//Error FB instances
EL5021_Error(
    En                  := TRUE,
    iTerminal_ID        := iTerminal_ID,
    bWcState            := WcState_WcState,
    uiInfoData_State    := InfoData_State,
    pErrorSystem        := ErrorSystem,
    bError => bError,
);

IF bError THEN
    sErrorMessage:=EL5021_Error.ErrorData.sErrorMessage;
ELSE
	sErrorMessage:='';
END_IF

END_FUNCTION_BLOCK

// ---- POUs/Common/Hardware/EtherCAT_Terminals/Communication/EL6695.TcPOU
//EL6695 | EtherCAT bridge termina
FUNCTION_BLOCK EL6695

VAR_INPUT
    En: BOOL;
    iTerminal_ID : INT;
    ErrorSystem : POINTER TO ST_ErrorSystem;
END_VAR

VAR_OUTPUT
    EnO: BOOL;
    bError: BOOL;
	sErrorMessage       : STRING;
END_VAR

VAR
    WcState_WcState AT %I* : BOOL := FALSE;
    InfoData_State  AT %I* : UINT := 0;

    //FB-s
    EL6695_Error    : FB_TerminalError;
END_VAR

(*
* TODO: Test on hardware
*)

EnO:=En;

EL6695_Error(
    En := TRUE,
    iTerminal_ID := iTerminal_ID,
    bWcState := FALSE,
    uiInfoData_State := InfoData_State,
    pErrorSystem := ErrorSystem,
    bError => bError,
);

IF bError THEN
	sErrorMessage:=EL6695_Error.ErrorData.sErrorMessage;
ELSE
	sErrorMessage:='';
END_IF

END_FUNCTION_BLOCK

// ---- POUs/Common/Hardware/EtherCAT_Terminals/Digital_Outputs/EL2032.TcPOU
// EL2032 | 2-channel digital output terminal 24 V DC, 2 A
FUNCTION_BLOCK EL2032

VAR_INPUT
    En: BOOL;
    iTerminal_ID : INT;
    ErrorSystem : POINTER TO ST_ErrorSystem;
END_VAR

VAR_OUTPUT
    EnO: BOOL;
    bError: BOOL;
	sErrorMessage       : STRING;
END_VAR

VAR
    WcState_WcState AT %I* : BOOL := FALSE;
    InfoData_State  AT %I* : UINT := 0;

    //FB-s
    EL2032_Error    : FB_TerminalError;
END_VAR

(*
* TODO: Test on hardware
*)

EnO:=En;

EL2032_Error(
    En := TRUE,
    iTerminal_ID := iTerminal_ID,
    bWcState := FALSE,
    uiInfoData_State := InfoData_State,
    pErrorSystem := ErrorSystem,
    bError => bError,
);

IF bError THEN
	sErrorMessage:=EL2032_Error.ErrorData.sErrorMessage;
ELSE
	sErrorMessage:='';
END_IF

END_FUNCTION_BLOCK

// ---- POUs/Common/Hardware/EtherCAT_Terminals/System/EK1110.TcPOU
FUNCTION_BLOCK EK1110

VAR_INPUT
    En              : BOOL;
    iTerminal_ID    : INT;
    ErrorSystem     : POINTER TO ST_ErrorSystem;
END_VAR

VAR_OUTPUT
    EnO     : BOOL;
    bError  : BOOL;
	sErrorMessage       : STRING;
END_VAR

VAR
    InfoData_State  AT %I*  : UINT;
    
    //FB-s
    EK1110_Error    : FB_TerminalError;
END_VAR

(*
* TODO: DONE!
*)
EnO:=En;

//Error FB instance
EK1110_Error(
    En                  := TRUE,
    iTerminal_ID        := iTerminal_ID,
    bWcState            := FALSE,
    uiInfoData_State    := InfoData_State,
    pErrorSystem        := ErrorSystem,
    bError              => bError,
);

IF bError THEN
	sErrorMessage:=EK1110_Error.ErrorData.sErrorMessage;
ELSE
	sErrorMessage:='';
END_IF

END_FUNCTION_BLOCK

// ---- POUs/Common/Hardware/EtherCAT_Terminals/Drives/indraDrive.TcPOU
//Rexroth indradrive
FUNCTION_BLOCK indraDrive

VAR_INPUT
    En: BOOL;
    iTerminal_ID : INT;
    ErrorSystem : POINTER TO ST_ErrorSystem;
END_VAR

VAR_OUTPUT
    EnO: BOOL;
    bError: BOOL;
	sErrorMessage       : STRING;
END_VAR

VAR
    WcState_WcState AT %I* : BOOL := FALSE;
    InfoData_State  AT %I* : UINT := 0;

    //FB-s
    indraDrive_Error    : FB_TerminalError;
END_VAR

(*
* TODO: Test on hardware
*)

EnO:=En;

indraDrive_Error(
    En := TRUE,
    iTerminal_ID := iTerminal_ID,
    bWcState := FALSE,
    uiInfoData_State := InfoData_State,
    pErrorSystem := ErrorSystem,
    bError => bError,
);

IF bError THEN
	sErrorMessage:=indraDrive_Error.ErrorData.sErrorMessage;
ELSE
	sErrorMessage:='';
END_IF

END_FUNCTION_BLOCK

// ---- POUs/Common/Hardware/EtherCAT_Terminals/Drives/iPOS8020.TcPOU
//Technosoft iPOS8020
FUNCTION_BLOCK iPOS8020

VAR_INPUT
    En: BOOL;
    iTerminal_ID : INT;
    ErrorSystem : POINTER TO ST_ErrorSystem;
END_VAR

VAR_OUTPUT
    EnO: BOOL;
    bError: BOOL;
	sErrorMessage       : STRING;
END_VAR

VAR
    WcState_WcState AT %I* : BOOL := FALSE;
    InfoData_State  AT %I* : UINT := 0;

    //FB-s
    iPOS8020_Error    : FB_TerminalError;
END_VAR

(*
* TODO: Test on hardware
*)

EnO:=En;

iPOS8020_Error(
    En := TRUE,
    iTerminal_ID := iTerminal_ID,
    bWcState := FALSE,
    uiInfoData_State := InfoData_State,
    pErrorSystem := ErrorSystem,
    bError => bError,
);

IF bError THEN
	sErrorMessage:=iPOS8020_Error.ErrorData.sErrorMessage;
ELSE
	sErrorMessage:='';
END_IF

END_FUNCTION_BLOCK

// ---- POUs/Bridge Terminal/TSCS_Bridge_Inputs.TcPOU
PROGRAM TSCS_Bridge_Inputs	
(* Inputs from TSCS PLC to TDU PLC*)
VAR
	// Function Blocks
	BYTE_TO_BITS_10: OSCAT_BYTE_TO_BITS; // Interface for TSCS Byte 0 - Boolean inputs
	BYTE_TO_BITS_11: OSCAT_BYTE_TO_BITS; // Interface for TSCS Byte 1 - Boolean inputs
	BYTE_TO_BITS_12: OSCAT_BYTE_TO_BITS; // Interface for TSCS Byte 2 - Boolean inputs
	BYTE_TO_BITS_13: OSCAT_BYTE_TO_BITS; // Interface for TSCS Byte 3 - Boolean inputs
	fb_Bridge_Real_Inputs_0 : FB_Bridge_Inputs_Real; // Interface for TSCS real signals
	fb_Bridge_Real_Inputs_1 : FB_Bridge_Inputs_Real; // Interface for TMS real signals
	
	// Test Signal
	TDU_TestSignal_RB : REAL;	// Diagnostic signal readback (TDU -> TSCS ->TDU)
		
	// TSCS signals (as example)
	Lube_MainBearing_Act : BOOL; 		// Main bearing lubrication active
	TSCS_State : INT; 					// Target System Operation Mode [0=Off, 1=Normal Operation, 2=Maintenance]
	Lube_MainBearing_FlowRate : REAL; 	// Main bearing lubrication flow rate [mL/min]
END_VAR

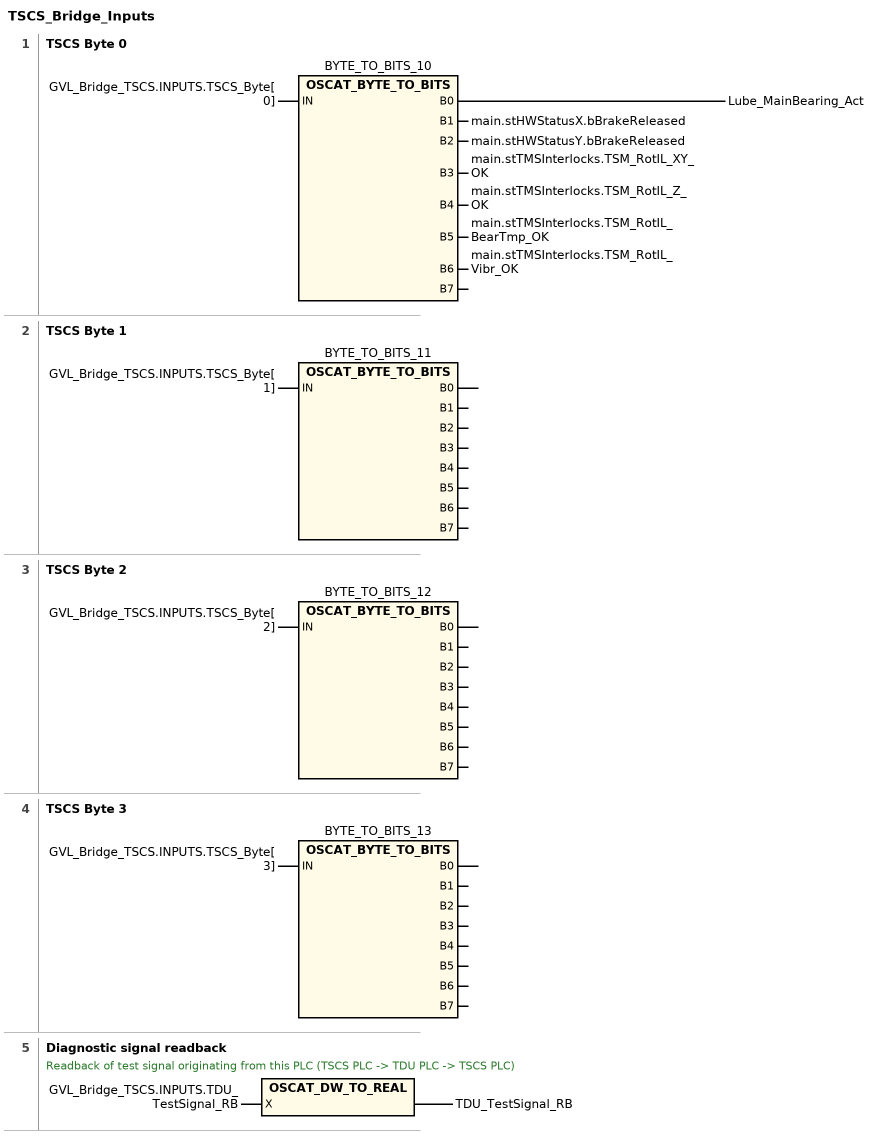
// NETWORK 1: TSCS Byte 0
BYTE_TO_BITS_10(
    IN := GVL_Bridge_TSCS.INPUTS.TSCS_Byte[0],
    B1 => main.stHWStatusX.bBrakeReleased,
    B2 => main.stHWStatusY.bBrakeReleased,
    B3 => main.stTMSInterlocks.TSM_RotIL_XY_OK,
    B4 => main.stTMSInterlocks.TSM_RotIL_Z_OK,
    B5 => main.stTMSInterlocks.TSM_RotIL_BearTmp_OK,
    B6 => main.stTMSInterlocks.TSM_RotIL_Vibr_OK); // OSCAT_BYTE_TO_BITS
Lube_MainBearing_Act := BYTE_TO_BITS_10.B0;

// NETWORK 2: TSCS Byte 1
BYTE_TO_BITS_11(IN := GVL_Bridge_TSCS.INPUTS.TSCS_Byte[1]); // OSCAT_BYTE_TO_BITS

// NETWORK 3: TSCS Byte 2
BYTE_TO_BITS_12(IN := GVL_Bridge_TSCS.INPUTS.TSCS_Byte[2]); // OSCAT_BYTE_TO_BITS

// NETWORK 4: TSCS Byte 3
BYTE_TO_BITS_13(IN := GVL_Bridge_TSCS.INPUTS.TSCS_Byte[3]); // OSCAT_BYTE_TO_BITS

// NETWORK 5: Diagnostic signal readback
// Readback of test signal originating from this PLC (TSCS PLC -> TDU PLC -> TSCS PLC)
TDU_TestSignal_RB := OSCAT_DW_TO_REAL(X := GVL_Bridge_TSCS.INPUTS.TDU_TestSignal_RB);

END_PROGRAM

// ---- POUs/Bridge Terminal/FBs/OSCAT_BYTE_TO_BITS.TcPOU
FUNCTION_BLOCK OSCAT_BYTE_TO_BITS
// E. Foy (2021-08-30): Copied from OSCAT library.
VAR_INPUT
	IN: BYTE;
END_VAR
VAR_OUTPUT
	B0: BOOL;
	B1: BOOL;
	B2: BOOL;
	B3: BOOL;
	B4: BOOL;
	B5: BOOL;
	B6: BOOL;
	B7: BOOL;
END_VAR


(*
version 1.1	16. mar. 2008
programmer 	hugo
tested by		tobias

this Function Block extracts the 8 Bits from a byte


*)

B0 := IN.0;
B1 := IN.1;
B2 := IN.2;
B3 := IN.3;
B4 := IN.4;
B5 := IN.5;
B6 := IN.6;
B7 := IN.7;

(* revision history
hm		4. aug 2006	rev 1.0
	original version

hm		16. mar 2008	rev 1.1
	renamed from byte_to_bit to byte_to_bits for compatibility reasons

*)

END_FUNCTION_BLOCK

// ---- POUs/Bridge Terminal/FBs/FB_Bridge_Inputs_Real.TcPOU
FUNCTION_BLOCK FB_Bridge_Inputs_Real
// Interface with 20 ports. Converts UDINT to REAL (32 bits)
VAR_INPUT
	I00 : UDINT := 0;	// Input real 00
	I01 : UDINT := 0;	// Input real 01
	I02 : UDINT := 0;	// Input real 02
	I03 : UDINT := 0;	// Input real 03
	I04 : UDINT := 0;	// Input real 04
	I05 : UDINT := 0;	// Input real 05
	I06 : UDINT := 0;	// Input real 06
	I07 : UDINT := 0;	// Input real 07
END_VAR
VAR_OUTPUT
	Q00 : REAL;
	Q01 : REAL;
	Q02 : REAL;
	Q03 : REAL;
	Q04 : REAL;
	Q05 : REAL;
	Q06 : REAL;
	Q07 : REAL;
END_VAR
VAR
END_VAR

Q00 := OSCAT_DW_TO_REAL(I00);
Q01 := OSCAT_DW_TO_REAL(I01);
Q02 := OSCAT_DW_TO_REAL(I02);
Q03 := OSCAT_DW_TO_REAL(I03);
Q04 := OSCAT_DW_TO_REAL(I04);
Q05 := OSCAT_DW_TO_REAL(I05);
Q06 := OSCAT_DW_TO_REAL(I06);
Q07 := OSCAT_DW_TO_REAL(I07);

END_FUNCTION_BLOCK

// ---- POUs/Bridge Terminal/FBs/OSCAT_DW_TO_REAL.TcPOU
FUNCTION OSCAT_DW_TO_REAL : REAL
// E. Foy (2021-08-30): Copied from OSCAT library.
VAR_INPUT
	X : DWORD;
END_VAR
VAR
	pt : POINTER TO REAL;
END_VAR

(*
version 1.0	18. apr. 2008
programmer 	hugo
tested by		tobias

this function converts a DWORD to REAL in a bitwise manner.
*)

pt := ADR(X);
OSCAT_DW_TO_REAL := pt^;

(* revision history
hm	18. apr. 2008
	original version

*)

END_FUNCTION

// ---- POUs/Bridge Terminal/TSCS_Bridge_Diagnostic.TcPOU
PROGRAM TSCS_Bridge_Diagnostic
(*Generates a test signal for the bridge terminal then compares it against a readback signal*)
VAR
	TestSignal : REAL;
	
	TDU_TestSignal_Delay :REAL := 0; // Number of counts behind the TDU TestSignal
	TMS_TestSignal_Delay :REAL := 0; // Number of counts behind the TMS TestSignal 
	
	// Parameters
	CountRate : REAL := 1.0; // ms per cycle (e.g. 1.0 for a 1ms excution rate)
	Signal_HL : REAL := 1000; // Signal High Limit
	Signal_LL : REAL := -1000; // Signal Low Limit
 
	RS_0: RS;	// Counter state (Set = Count-DOWN active)
END_VAR
VAR // added by the converter: edge detectors and wires of the graphical bodies
    _rt1, _rt2 : R_TRIG;
END_VAR

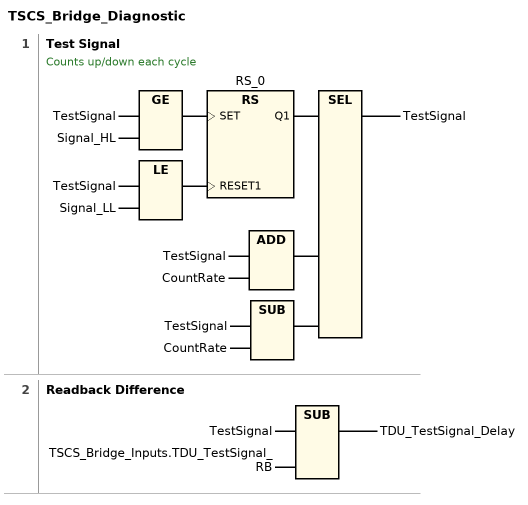
// NETWORK 1: Test Signal
// Counts up/down each cycle
_rt1(CLK := TestSignal >= Signal_HL);
_rt2(CLK := TestSignal <= Signal_LL);
RS_0(SET := _rt1.Q, RESET1 := _rt2.Q); // RS
TestSignal := SEL(RS_0.Q1, TestSignal + CountRate, TestSignal - CountRate);

// NETWORK 2: Readback Difference
TDU_TestSignal_Delay := TestSignal - TSCS_Bridge_Inputs.TDU_TestSignal_RB;

END_PROGRAM

// ---- POUs/Bridge Terminal/TSCS_Bridge_Outputs.TcPOU
PROGRAM TSCS_Bridge_Outputs
(*Outputs from TDU PLC to TSCS PLC*)
VAR
	// Function Blocks
	fb_Bridge_Outputs_Real_0 : FB_Bridge_Outputs_Real; // Interface for TDU real outputs
	
	// Signal Conversions
	rActPos : REAL; // Rotation system - Actual Position [deg]
	rActVel : REAL; // Rotation system - Actual Velocity [rpm]
	rSetVelRaw : REAL; //Rotation system - Velocity setpoint raw [rpm] 
	
END_VAR

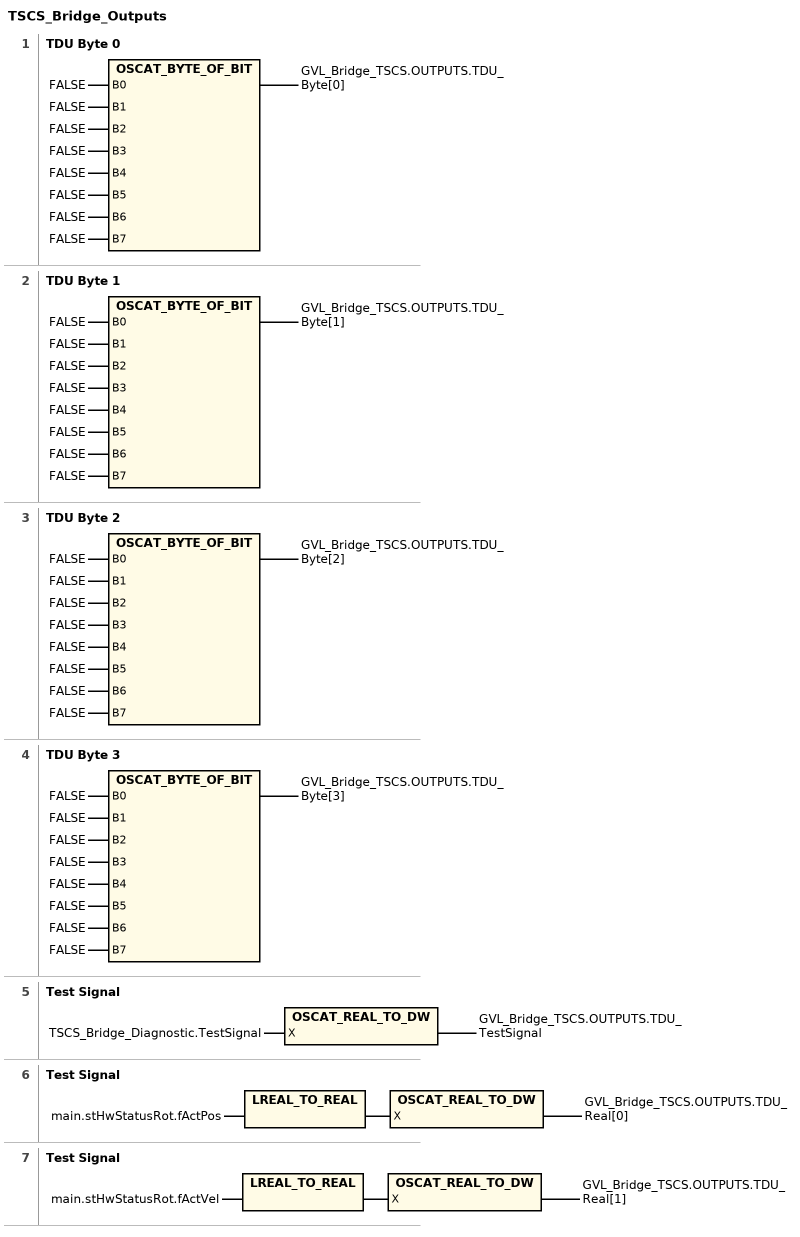
// NETWORK 1: TDU Byte 0
GVL_Bridge_TSCS.OUTPUTS.TDU_Byte[0] := OSCAT_BYTE_OF_BIT(B0 := FALSE, B1 := FALSE, B2 := FALSE, B3 := FALSE, B4 := FALSE, B5 := FALSE, B6 := FALSE, B7 := FALSE);

// NETWORK 2: TDU Byte 1
GVL_Bridge_TSCS.OUTPUTS.TDU_Byte[1] := OSCAT_BYTE_OF_BIT(B0 := FALSE, B1 := FALSE, B2 := FALSE, B3 := FALSE, B4 := FALSE, B5 := FALSE, B6 := FALSE, B7 := FALSE);

// NETWORK 3: TDU Byte 2
GVL_Bridge_TSCS.OUTPUTS.TDU_Byte[2] := OSCAT_BYTE_OF_BIT(B0 := FALSE, B1 := FALSE, B2 := FALSE, B3 := FALSE, B4 := FALSE, B5 := FALSE, B6 := FALSE, B7 := FALSE);

// NETWORK 4: TDU Byte 3
GVL_Bridge_TSCS.OUTPUTS.TDU_Byte[3] := OSCAT_BYTE_OF_BIT(B0 := FALSE, B1 := FALSE, B2 := FALSE, B3 := FALSE, B4 := FALSE, B5 := FALSE, B6 := FALSE, B7 := FALSE);

// NETWORK 5: Test Signal
GVL_Bridge_TSCS.OUTPUTS.TDU_TestSignal := OSCAT_REAL_TO_DW(X := TSCS_Bridge_Diagnostic.TestSignal);

// NETWORK 6: Test Signal
GVL_Bridge_TSCS.OUTPUTS.TDU_Real[0] := OSCAT_REAL_TO_DW(X := LREAL_TO_REAL(main.stHwStatusRot.fActPos));

// NETWORK 7: Test Signal
GVL_Bridge_TSCS.OUTPUTS.TDU_Real[1] := OSCAT_REAL_TO_DW(X := LREAL_TO_REAL(main.stHwStatusRot.fActVel));

END_PROGRAM

// ---- POUs/Bridge Terminal/FBs/FB_Bridge_Outputs_Real.TcPOU
FUNCTION_BLOCK FB_Bridge_Outputs_Real
// Interface with 20 ports. Converts REAL to UDINT (32 bits)
VAR_INPUT
	I00 : REAL := 0;
	I01 : REAL := 0;
	I02 : REAL := 0;
	I03 : REAL := 0;
	I04 : REAL := 0;
	I05 : REAL := 0;
	I06 : REAL := 0;
	I07 : REAL := 0;
END_VAR
VAR_OUTPUT
	Q00 : UDINT;
	Q01 : UDINT;
	Q02 : UDINT;
	Q03 : UDINT;
	Q04 : UDINT;
	Q05 : UDINT;
	Q06 : UDINT;
	Q07 : UDINT;
END_VAR
VAR
END_VAR

Q00 := OSCAT_REAL_TO_DW(I00);
Q01 := OSCAT_REAL_TO_DW(I01);
Q02 := OSCAT_REAL_TO_DW(I02);
Q03 := OSCAT_REAL_TO_DW(I03);
Q04 := OSCAT_REAL_TO_DW(I04);
Q05 := OSCAT_REAL_TO_DW(I05);
Q06 := OSCAT_REAL_TO_DW(I06);
Q07 := OSCAT_REAL_TO_DW(I07);

END_FUNCTION_BLOCK

// ---- POUs/Bridge Terminal/FBs/OSCAT_REAL_TO_DW.TcPOU
FUNCTION OSCAT_REAL_TO_DW : DWORD
// E. Foy (2021-08-30): Copied from OSCAT library.
VAR_INPUT
	X : REAL;
END_VAR
VAR
	pt : POINTER TO DWORD;
END_VAR

(*
version 1.0	18. apr. 2008
programmer 	hugo
tested by		tobias

this function converts a 32 Bit Real to a dword in a bitwise manner.
*)

pt := ADR(X);
OSCAT_REAL_TO_DW := pt^;

(* revision history
hm	18. apr. 2008
	original version

*)

END_FUNCTION

// ---- POUs/Bridge Terminal/FBs/OSCAT_BYTE_OF_BIT.TcPOU
FUNCTION OSCAT_BYTE_OF_BIT : BYTE
// E. Foy (2021-08-30): Copied from OSCAT library.
VAR_INPUT
	B0:BOOL;
	B1:BOOL;
	B2:BOOL;
	B3:BOOL;
	B4:BOOL;
	B5:BOOL;
	B6:BOOL;
	B7:BOOL;
END_VAR

(*
version 1.1	 18. feb 2006
programmer 	hugo
tested by		tobias

this function creates a byte from 8 individual bits

*)

OSCAT_BYTE_OF_BIT := SHL(SHL(SHL(SHL(SHL(SHL(SHL(BOOL_TO_BYTE(B7),1) OR BOOL_TO_BYTE(B6),1) OR BOOL_TO_BYTE(B5),1) OR BOOL_TO_BYTE(B4),1)
	OR BOOL_TO_BYTE(B3),1) OR BOOL_TO_BYTE(B2),1) OR BOOL_TO_BYTE(B1),1) OR BOOL_TO_BYTE(B0);


(* revision history

hm	4. aug 2006		rev 1.0
	original version

hm	18. feb. 2008	rev 1.1
	improved performance

*)

END_FUNCTION

// ---- POUs/MAIN_NORMAL_MOTION.TcPOU
PROGRAM MAIN_NORMAL_MOTION
VAR
    sVersion: STRING := '1.0.0';

    //hmiAxisSelection: INT := 1; //Not possible to use local hmi variables for array indexes

//Startup, Shutdown and UPS
    fbUPS: FB_S_UPS_CX51x0;
    eUpsMode: E_S_UPS_Mode := eSUPS_WrPersistData_Shutdown;
    eStartUp: (eColdStart, eReadAxisFeedbackType, eCheckReadDone, eExecuteRestore, eCheckRestore, eFinishRestore);
    bPositionRestoreDone: BOOL := FALSE;
    bRestoreExecute: BOOL := FALSE;
    bExecuteReadEncRefSys: BOOL := FALSE;
    nRetry: INT;
    iAxes : UINT; //index for for loops in Position recovery actions
    afbReadEncRefSys: ARRAY [1..GVL_APP.nAXIS_NUM] OF MC_ReadParameter;
    afbRestorePosition: ARRAY [1..GVL_APP.nAXIS_NUM] OF MC_SetPosition;
    fbGetDeviceIdentification: FB_GetDeviceIdentification;
END_VAR

VAR PERSISTENT
    bRestoreOnStartup: BOOL;
END_VAR

// Block PILS
GVL.bLocalMode:=TRUE;

POSITION_RECOVERY();
AXES();
PROG();

ACTION AXES:
//Get task index for Axes parameters initialization.
GVL.fbGetCurTaskIndex();

//Create an stAxisStruct for every axis in the project.
FOR GVL.iAxis := 1 TO GVL_APP.nAXIS_NUM DO
    Main.afbAxes[GVL.iAxis](stAxisStruct := GVL.astAxes[GVL.iAxis]);
END_FOR
END_ACTION

ACTION CHECK_UPS:
fbUPS(eUpsMode := eUpsMode);

IF eGlobalSUpsState = eSUPS_PowerFailure THEN
    //first cycle of powerfailure
    //execute code that should only be done once with each powerfailure, i.e. increase powerfailure counter
    bRestoreOnStartup := TRUE;
    STORE_PERSISTENT();
    RETURN;
ELSIF eGlobalSUpsState <> eSUPS_PowerOK THEN
    //next cycles of powerfailure
    //skip regular code execution for the remaining cycles of the powerfailure/writing of persistent data/quick shutdown...
    RETURN;
END_IF
END_ACTION

ACTION POSITION_RECOVERY:
fbGetDeviceIdentification(bExecute := TRUE);
IF (fbGetDeviceIdentification.stDevIdent.strHardwareSerialNo <> '0') THEN
    CHECK_UPS();
    RESTORE_POSITIONS();
END_IF
END_ACTION

ACTION PROG:
//Call the programs that are defined in the "Application Specific" folder.
//Create as many programs in that folder as axes and applications you have or need

//Axes initial parameters and program
//Axis_Template();
Axis_1();
Axis_2();
Axis_3();

//Application program calls
//Application_Template();
END_ACTION

ACTION RESTORE_POSITIONS:
//This ACT will restore the position of an incremental axis on startup with the act position it read before losing power.
//It checks the type of axis, 0=incremental, and that the axis was stationary at shut down.
//Because 0 equates to incremental we also need to check that the data is valid, otherwise by default it would restore all axes.
//By default an axis will not restore the position unless it is set to opt-in, i.e. GVL.aAxes[iAxes].stConfig.eRestorePosition is non-zero.
//This needs to be initialised somewhere in TwinCAT code otherwise it will not be available at start up.
//A restore will only be performed on a loss of power, this code shouldn't make any changes on a reset cold, a rest origin or a download.
//There is a enum to allow for different types of restore modes, currently only one is implemented.
//0 'DontRestore'
//1 'RestoreWithoutHome' -restores the position using a set position fb and does not set the home bit in the axis struct.
//Note from Beckhoff: "A maximum of 1 MB persistent data can be reliably saved over the entire service life."

IF bRestoreOnStartup AND eGlobalSUpsState = eSUPS_PowerOK THEN
    bRestoreOnStartup := FALSE;
    bRestoreExecute := TRUE;
END_IF

//Upon startup bPositionRestoreDone will be set to FALSE, after successfully completing the following code it will be set TRUE
//and should stay TRUE for the rest of the time the PLC is operational, thus this routine should only be completed once.
IF bRestoreExecute AND NOT bPositionRestoreDone THEN
    //Cycle through function blocks that read the encoder reference system i.e. whether axis is incremental or absolute
    //Result stored in Value, 0=Inc 1=Abs, execute set during the case statement
    FOR iAxes := 1 TO GVL_APP.nAXIS_NUM DO
        afbReadEncRefSys[iAxes](
          Axis := GVL.astAxes[iAxes].Axis,
          Enable := bExecuteReadEncRefSys,
          ParameterNumber := MC_AxisParameter.AxisEncoderReferenceSystem,
          ReadMode := E_READMODE.READMODE_ONCE);
    END_FOR

    //Cycle through set position function blocks for each axis
    FOR iAxes := 1 TO GVL_APP.nAXIS_NUM DO
        afbRestorePosition[iAxes](
         Axis := GVL.astAxes[iAxes].Axis,
         Position := astAxesPersistent[iAxes].fPositionAtShutdown);
    END_FOR

    CASE eStartUp OF
        eColdStart:
        //First cycle of the PLC, do nothing just give one cycle for variables to initialise
            IF NOT bPositionRestoreDone THEN
                eStartUp := eReadAxisFeedbackType;
                nRetry := 0;
            END_IF

        eReadAxisFeedbackType:
        //Exectute the function blocks to read the encoder reference system (0=inc OR 1=ABS)
            bExecuteReadEncRefSys := TRUE;
            eStartUp := eCheckReadDone;

        eCheckReadDone:
        //Check the encoder reference system has been read for all axis -> if busy then continue with PLC cycle and check again next time.
        //If afbReadEncRefSys not started then go back a step.
        //If any axes result in an error the code will get stuck here, this happens if GVL_APP.nAXIS_NUM is not set correctly
            FOR iAxes := 1 TO GVL_APP.nAXIS_NUM DO
                IF afbReadEncRefSys[iAxes].Valid = FALSE THEN
                    IF afbReadEncRefSys[iAxes].Busy = TRUE THEN
                        //Exit MAIN.STARTUP Action and wait till next cycle, needs to cycle through whole program in order for data to update
                        RETURN;
                    ELSE
                        //Sometimes the code gets here and the afbReadEncRefSys[iAxes] misses the rising edge. If  the code gets here it means
                        //valid=FALSE and .busy=FALSE which indicateds the FB probably hasn't started and thus needs to see a rising edge.
                        //Set execute to low, Exit MAIN.STARTUP and go back a step in the CASE statement.
                        bExecuteReadEncRefSys := FALSE;
                        eStartUp := eReadAxisFeedbackType;
                        nRetry := nRetry + 1; //counter used for troubleshooting to see how many cycles it takes before afbReadEncRefSys function blocks are read correctly
                        RETURN;
                    END_IF
                END_IF
            END_FOR
            //If the code gets here all axes either have .valid=TRUE for all axes
            eStartUp := eExecuteRestore;

        eExecuteRestore:
        //Execute position restore by setting afbRestorePosition.execute = TRUE
            FOR iAxes := 1 TO GVL_APP.nAXIS_NUM DO
                IF afbReadEncRefSys[iAxes].Valid = TRUE AND afbReadEncRefSys[iAxes].Value = 0 AND NOT(astAxesPersistent[iAxes].bMovingAtShutdown) THEN
                    IF GVL.astAxes[iAxes].stConfig.eRestorePosition = E_RestorePosition.eRestoreWithoutHome THEN
                        afbRestorePosition[iAxes].Execute := TRUE;
                    END_IF
                END_IF
            END_FOR
            eStartUp := eCheckRestore;

        eCheckRestore:
        //Check the set position fbs are finished
        //Nothing actually happens if the restore is not done, the code just returns from here each cycle and the
        //bPositionRestoreDone will never get set to TRUE and will take up cycle time
            FOR iAxes := 1 TO GVL_APP.nAXIS_NUM DO
                IF afbReadEncRefSys[iAxes].Valid = TRUE AND afbReadEncRefSys[iAxes].Value = 0 AND NOT(astAxesPersistent[iAxes].bMovingAtShutdown) THEN
                    IF GVL.astAxes[iAxes].stConfig.eRestorePosition = E_RestorePosition.eRestoreWithoutHome THEN
                        IF NOT afbRestorePosition[iAxes].Done THEN
                            RETURN;
                        END_IF
                    END_IF
                END_IF
            END_FOR
            eStartUp := eFinishRestore;

        eFinishRestore:
        //Remove execute = TRUE for afbRestorePosition
            FOR iAxes := 1 TO GVL_APP.nAXIS_NUM DO
                afbRestorePosition[iAxes].Execute := FALSE;
            END_FOR
            bPositionRestoreDone := TRUE;
            bRestoreExecute := FALSE;
    END_CASE
END_IF
END_ACTION

ACTION STORE_PERSISTENT:
FOR iAxes := 1 TO GVL_APP.nAXIS_NUM DO
    astAxesPersistent[iAxes].fPositionAtShutdown := GVL.astAxes[iAxes].Axis.NcToPlc.ActPos;
    IF GVL.astAxes[iAxes].Axis.NcToPlc.ActVelo <> 0 THEN
        astAxesPersistent[iAxes].bMovingAtShutdown := TRUE;
    ELSE
        astAxesPersistent[iAxes].bMovingAtShutdown := FALSE;
    END_IF
    astAxesPersistent[iAxes].bMovingAtShutdown := astAxesPersistent[iAxes].bMovingAtShutdown OR GVL.astAxes[iAxes].Axis.Status.Moving;
END_FOR
END_ACTION

END_PROGRAM

// ---- POUs/Application_Specific/Axes/Axis_1.TcPOU
PROGRAM Axis_1
VAR
    bLimitPowerAxis1 AT %Q*: BOOL := TRUE;
END_VAR
VAR // added by the converter: edge detectors and wires of the graphical bodies
    _w1, _w2 : BOOL;
END_VAR

//Initial parameters of an Axis
IF _TaskInfo[fbGetCurTaskIndex.index].FirstCycle THEN
    //Initial default values:
    GVL.astAxes[1].stConfig.eHomeSeq := 0;
    GVL.astAxes[1].stConfig.fHomePosition := 0.0;
    GVL.astAxes[1].stConfig.fHomeFinishDistance := 0.0;
END_IF

ACT_1_Interlock();

// Brake control from GUI
// main.stHWStatusX.bBrakeReleased:=main.stHWControlX.bBrakeReleaseCmd;

// Enable Cmd from GUI
GVL.astAxes[1].stControl.bEnable:=main.stHWControlX.bEnable;
main.stHWStatusX.bEnabled:=GVL.astAxes[1].stStatus.bEnabled;

// Trigger Abs movement from GUI
IF main.stHWControlX.bExecuteAbsPos  AND NOT GVL.astAxes[1].stStatus.bBusy THEN
  GVL.astAxes[1].stControl.eCommand:=E_MotionFunctions.eMoveAbsolute;
  GVL.astAxes[1].stControl.bExecute:=TRUE;
  main.stHWControlX.bExecuteAbsPos:=FALSE;
END_IF

// Trigger Const Velo movement from GUI
IF main.stHWControlX.bExecuteConstVelo AND NOT GVL.astAxes[1].stStatus.bBusy THEN
  GVL.astAxes[1].stControl.eCommand:=E_MotionFunctions.eMoveVelocity;
  GVL.astAxes[1].stControl.bExecute:=TRUE;
  main.stHWControlX.bExecuteConstVelo:=FALSE;
END_IF

// Trigger Home vs LimitFwd (should be valid for all axes) from GUI
IF main.stHWControlX.bExecuteHome  AND NOT GVL.astAxes[1].stStatus.bBusy THEN
  GVL.astAxes[1].stConfig.fHomingVelFromCam:=GVL_Parameters.fXHomeVelOffCam;
  GVL.astAxes[1].stConfig.fHomingVelToCam:=GVL_Parameters.fXHomeVelToCam;
  GVL.astAxes[1].stConfig.fHomePosition:=GVL_Parameters.fXHomePosition;
  GVL.astAxes[1].stControl.eCommand:=E_MotionFunctions.eHome;
  GVL.astAxes[1].stConfig.eHomeSeq:=E_HomingRoutines.eHomeToLimit_Fwd;
  GVL.astAxes[1].stControl.bExecute:=TRUE;
  main.stHWControlX.bExecuteHome:=FALSE;
END_IF

//Stop Motion from GUI
IF main.stHWControlX.bExecuteStop THEN
  GVL.astAxes[1].stControl.bStop := NOT(GVL.astAxes[1].stControl.bStop);
  GVL.astAxes[1].stControl.bExecute:=FALSE;
  main.stHWControlX.bExecuteStop:=FALSE;
END_IF

// Error Code
GVL.astAxes[1].stStatus.nErrorID;

main.stHWStatusX.bBusy:=GVL.astAxes[1].stStatus.bBusy;
GVL.astAxes[1].stControl.bReset:=main.stHWControlX.bExecuteReset;
main.stHWControlX.bExecuteReset:=FALSE;
main.stHWStatusX.bHomed:=GVL.astAxes[1].stStatus.bHomed;
main.stHWStatusX.bHomingCmdActive:=GVL.astAxes[1].stControl.eCommand=E_MotionFunctions.eHome AND 
                                   GVL.astAxes[1].stConfig.eHomeSeq=E_HomingRoutines.eHomeToLimit_Fwd;

// Hard code velocities and acc/dec
GVL.astAxes[1].stControl.fAcceleration:=GVL_Parameters.fXStepperTargetAcc;
GVL.astAxes[1].stControl.fDeceleration:=GVL_Parameters.fXStepperTargetAcc;
GVL.astAxes[1].stControl.fVelocity:=GVL_Parameters.fXStepperTargetVelo;

// reverse velo if dir is BWD
IF GVL.astAxes[1].stControl.eCommand=E_MotionFunctions.eMoveVelocity AND NOT main.stHWControlX.bJogDirFwd  THEN
	GVL.astAxes[1].stControl.fVelocity:=-GVL_Parameters.fXStepperTargetVelo;
END_IF

// Check position is inside limits (and homed)
main.stHWStatusX.bLoLoAlm:=gvl.astAxes[1].stStatus.fActPosition < GVL_Parameters.fXRangeL2 OR NOT main.stHWStatusX.bHomed;
main.stHWStatusX.bLoAlm:=gvl.astAxes[1].stStatus.fActPosition < GVL_Parameters.fXRangeL1 OR NOT main.stHWStatusX.bHomed;
main.stHWStatusX.bHiAlm:=gvl.astAxes[1].stStatus.fActPosition > GVL_Parameters.fXRangeH1 OR NOT main.stHWStatusX.bHomed;
main.stHWStatusX.bhiHiAlm:=gvl.astAxes[1].stStatus.fActPosition > GVL_Parameters.fXRangeH2 OR NOT main.stHWStatusX.bHomed;

ACTION ACT_1_Interlock:
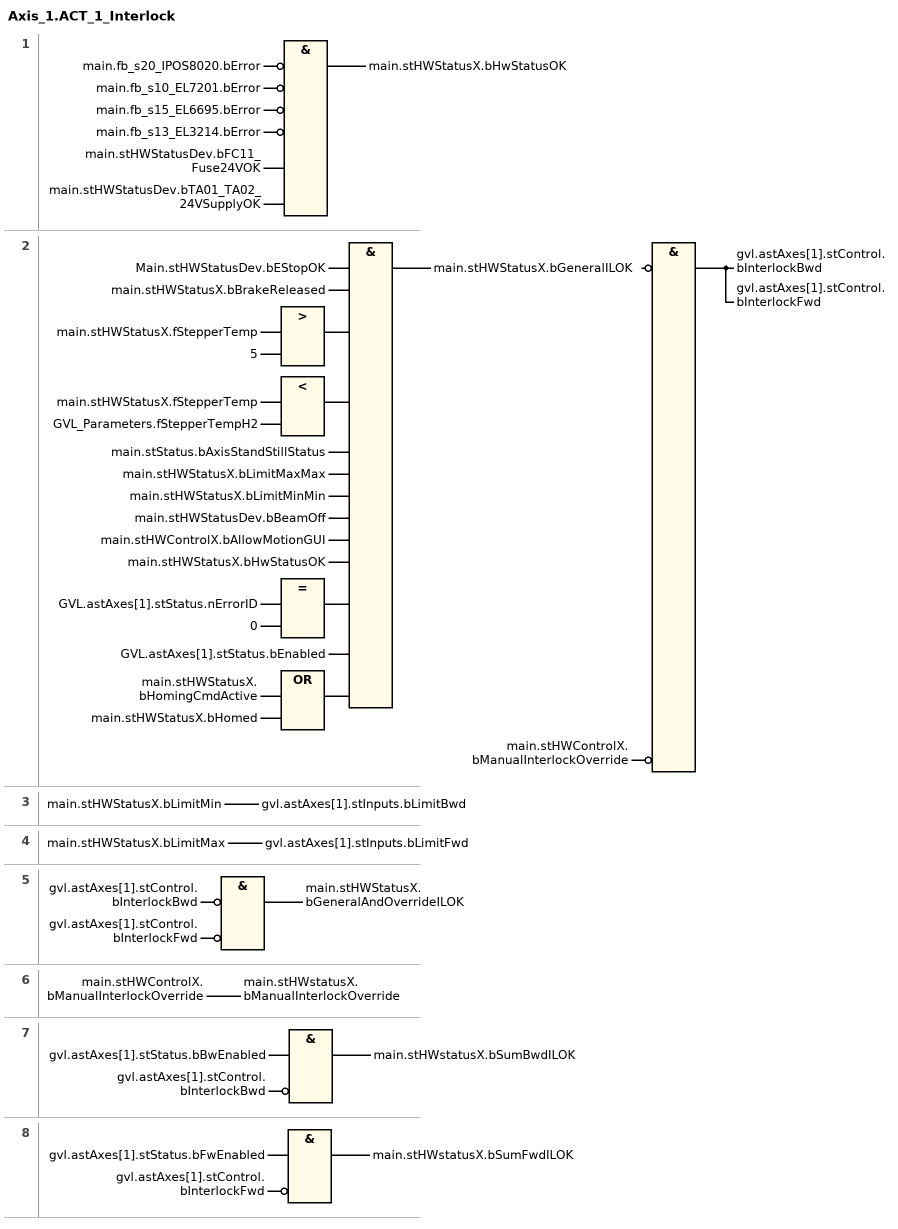
// NETWORK 1
main.stHWStatusX.bHwStatusOK := NOT main.fb_s20_IPOS8020.bError AND NOT main.fb_s10_EL7201.bError AND NOT main.fb_s15_EL6695.bError AND NOT main.fb_s13_EL3214.bError AND main.stHWStatusDev.bFC11_Fuse24VOK AND main.stHWStatusDev.bTA01_TA02_24VSupplyOK;

// NETWORK 2
_w1 := Main.stHWStatusDev.bEStopOK AND main.stHWStatusX.bBrakeReleased AND main.stHWStatusX.fStepperTemp > 5 AND main.stHWStatusX.fStepperTemp < GVL_Parameters.fStepperTempH2 AND main.stStatus.bAxisStandStillStatus AND main.stHWStatusX.bLimitMaxMax AND main.stHWStatusX.bLimitMinMin AND main.stHWStatusDev.bBeamOff AND main.stHWControlX.bAllowMotionGUI AND main.stHWStatusX.bHwStatusOK AND GVL.astAxes[1].stStatus.nErrorID = 0 AND GVL.astAxes[1].stStatus.bEnabled AND (main.stHWStatusX.bHomingCmdActive OR main.stHWStatusX.bHomed);
main.stHWStatusX.bGeneralILOK := _w1;
_w2 := NOT _w1 AND NOT main.stHWControlX.bManualInterlockOverride;
gvl.astAxes[1].stControl.bInterlockBwd := _w2;
gvl.astAxes[1].stControl.bInterlockFwd := _w2;

// NETWORK 3
gvl.astAxes[1].stInputs.bLimitBwd := main.stHWStatusX.bLimitMin;

// NETWORK 4
gvl.astAxes[1].stInputs.bLimitFwd := main.stHWStatusX.bLimitMax;

// NETWORK 5
main.stHWStatusX.bGeneralAndOverrideILOK := NOT gvl.astAxes[1].stControl.bInterlockBwd AND NOT gvl.astAxes[1].stControl.bInterlockFwd;

// NETWORK 6
main.stHWstatusX.bManualInterlockOverride := main.stHWControlX.bManualInterlockOverride;

// NETWORK 7
main.stHWstatusX.bSumBwdILOK := gvl.astAxes[1].stStatus.bBwEnabled AND NOT gvl.astAxes[1].stControl.bInterlockBwd;

// NETWORK 8
main.stHWstatusX.bSumFwdILOK := gvl.astAxes[1].stStatus.bFwEnabled AND NOT gvl.astAxes[1].stControl.bInterlockFwd;

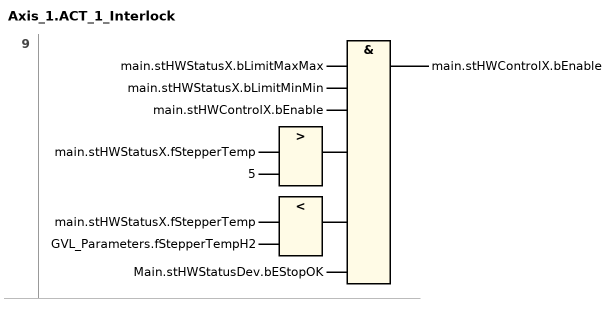
// NETWORK 9
main.stHWControlX.bEnable := main.stHWStatusX.bLimitMaxMax AND main.stHWStatusX.bLimitMinMin AND main.stHWControlX.bEnable AND main.stHWStatusX.fStepperTemp > 5 AND main.stHWStatusX.fStepperTemp < GVL_Parameters.fStepperTempH2 AND Main.stHWStatusDev.bEStopOK;
END_ACTION

END_PROGRAM

// ---- POUs/Application_Specific/Axes/Axis_2.TcPOU
PROGRAM Axis_2
VAR
	bLimitPowerAxis2 AT %Q*: BOOL := TRUE;
END_VAR
VAR // added by the converter: edge detectors and wires of the graphical bodies
    _w1, _w2 : BOOL;
END_VAR

//Initial parameters of an Axis
IF _TaskInfo[fbGetCurTaskIndex.index].FirstCycle THEN
    //Initial default values:
    GVL.astAxes[2].stConfig.eHomeSeq := 1;
    GVL.astAxes[2].stConfig.fHomePosition := 0.0;
    GVL.astAxes[2].stConfig.fHomeFinishDistance := 0;
END_IF

ACT_2_Interlock();

// Brake control from GUI
//main.stHWStatusY.bBrakeReleased:=main.stHWControlY.bBrakeReleaseCmd;

// Enable Cmd from GUI
GVL.astAxes[2].stControl.bEnable:=main.stHWControlY.bEnable;
main.stHWStatusY.bEnabled:=GVL.astAxes[2].stStatus.bEnabled;

// Trigger Abs movement from GUI
IF main.stHWControlY.bExecuteAbsPos  AND NOT GVL.astAxes[2].stStatus.bBusy THEN
  GVL.astAxes[2].stControl.eCommand:=E_MotionFunctions.eMoveAbsolute;
  GVL.astAxes[2].stControl.bExecute:=TRUE;
  main.stHWControlY.bExecuteAbsPos:=FALSE;
END_IF

// Trigger Const Velo movement from GUI
IF main.stHWControlY.bExecuteConstVelo AND NOT GVL.astAxes[2].stStatus.bBusy THEN
  GVL.astAxes[2].stControl.eCommand:=E_MotionFunctions.eMoveVelocity;
  GVL.astAxes[2].stControl.bExecute:=TRUE;
  main.stHWControlY.bExecuteConstVelo:=FALSE;
END_IF

// Trigger Home vs LimitFwd (should be valid for all axes) from GUI
IF main.stHWControlY.bExecuteHome  AND NOT GVL.astAxes[2].stStatus.bBusy THEN
  GVL.astAxes[2].stConfig.fHomePosition:=GVL_Parameters.fYHomePosition;
  GVL.astAxes[2].stConfig.fHomingVelFromCam:=GVL_Parameters.fYHomeVelOffCam;
  GVL.astAxes[2].stConfig.fHomingVelToCam:=GVL_Parameters.fYHomeVelToCam;
  GVL.astAxes[2].stControl.eCommand:=E_MotionFunctions.eHome;
  GVL.astAxes[2].stConfig.eHomeSeq:=E_HomingRoutines.eHomeToLimit_Fwd;
  GVL.astAxes[2].stControl.bExecute:=TRUE;
  main.stHWControlY.bExecuteHome:=FALSE;
END_IF

//Stop Motion from GUI
IF main.stHWControlY.bExecuteStop THEN
  GVL.astAxes[2].stControl.bStop := NOT(GVL.astAxes[2].stControl.bStop);
  GVL.astAxes[2].stControl.bExecute:=FALSE;
  main.stHWControlY.bExecuteStop:=FALSE;
END_IF

main.stHWStatusY.bBusy:=GVL.astAxes[2].stStatus.bBusy;
GVL.astAxes[2].stControl.bReset:=main.stHWControlY.bExecuteReset;
main.stHWControlY.bExecuteReset:=FALSE;
main.stHWStatusY.bHomed:=GVL.astAxes[2].stStatus.bHomed;
main.stHWStatusY.bHomingCmdActive:=GVL.astAxes[2].stControl.eCommand=E_MotionFunctions.eHome AND 
                                   GVL.astAxes[2].stConfig.eHomeSeq=E_HomingRoutines.eHomeToLimit_Fwd;

// Hard code velocities and acc/dec
GVL.astAxes[2].stControl.fAcceleration:=GVL_Parameters.fYStepperTargetAcc;
GVL.astAxes[2].stControl.fDeceleration:=GVL_Parameters.fYStepperTargetAcc;
GVL.astAxes[2].stControl.fVelocity:=GVL_Parameters.fYStepperTargetVelo;

// reverse velo if dir is BWD
IF GVL.astAxes[2].stControl.eCommand=E_MotionFunctions.eMoveVelocity AND NOT main.stHWControlY.bJogDirFwd  THEN
	GVL.astAxes[2].stControl.fVelocity:=-GVL_Parameters.fYStepperTargetVelo;
END_IF

// Check position is inside limits (and homed)
main.stHWStatusY.bLoLoAlm:=gvl.astAxes[2].stStatus.fActPosition < GVL_Parameters.fYRangeL2 OR NOT main.stHWStatusY.bHomed;
main.stHWStatusY.bLoAlm:=gvl.astAxes[2].stStatus.fActPosition < GVL_Parameters.fYRangeL1 OR NOT main.stHWStatusY.bHomed;;
main.stHWStatusY.bHiAlm:=gvl.astAxes[2].stStatus.fActPosition > GVL_Parameters.fYRangeH1 OR NOT main.stHWStatusY.bHomed;;
main.stHWStatusY.bhiHiAlm:=gvl.astAxes[2].stStatus.fActPosition > GVL_Parameters.fYRangeH2 OR NOT main.stHWStatusY.bHomed;;

ACTION ACT_2_Interlock:
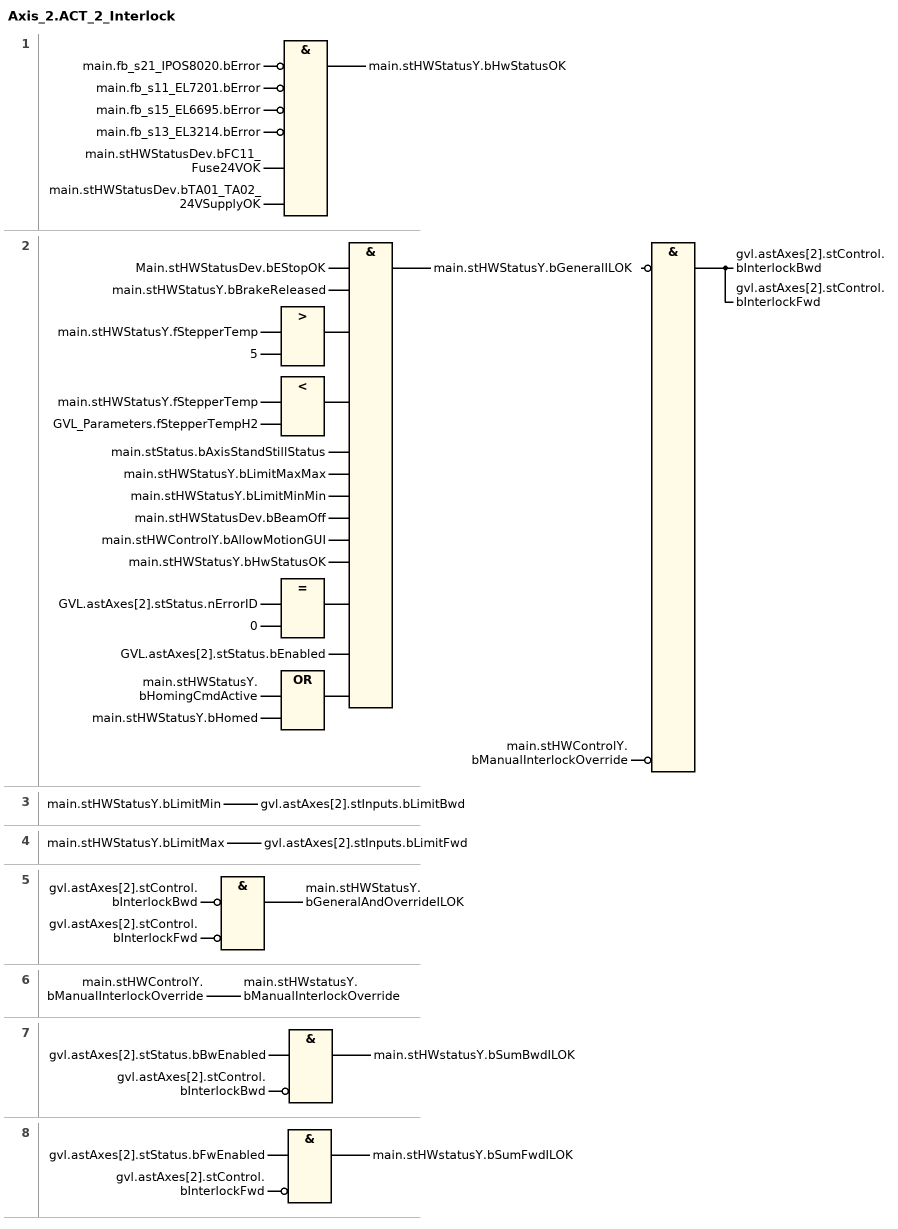
// NETWORK 1
main.stHWStatusY.bHwStatusOK := NOT main.fb_s21_IPOS8020.bError AND NOT main.fb_s11_EL7201.bError AND NOT main.fb_s15_EL6695.bError AND NOT main.fb_s13_EL3214.bError AND main.stHWStatusDev.bFC11_Fuse24VOK AND main.stHWStatusDev.bTA01_TA02_24VSupplyOK;

// NETWORK 2
_w1 := Main.stHWStatusDev.bEStopOK AND main.stHWStatusY.bBrakeReleased AND main.stHWStatusY.fStepperTemp > 5 AND main.stHWStatusY.fStepperTemp < GVL_Parameters.fStepperTempH2 AND main.stStatus.bAxisStandStillStatus AND main.stHWStatusY.bLimitMaxMax AND main.stHWStatusY.bLimitMinMin AND main.stHWStatusDev.bBeamOff AND main.stHWControlY.bAllowMotionGUI AND main.stHWStatusY.bHwStatusOK AND GVL.astAxes[2].stStatus.nErrorID = 0 AND GVL.astAxes[2].stStatus.bEnabled AND (main.stHWStatusY.bHomingCmdActive OR main.stHWStatusY.bHomed);
main.stHWStatusY.bGeneralILOK := _w1;
_w2 := NOT _w1 AND NOT main.stHWControlY.bManualInterlockOverride;
gvl.astAxes[2].stControl.bInterlockBwd := _w2;
gvl.astAxes[2].stControl.bInterlockFwd := _w2;

// NETWORK 3
gvl.astAxes[2].stInputs.bLimitBwd := main.stHWStatusY.bLimitMin;

// NETWORK 4
gvl.astAxes[2].stInputs.bLimitFwd := main.stHWStatusY.bLimitMax;

// NETWORK 5
main.stHWStatusY.bGeneralAndOverrideILOK := NOT gvl.astAxes[2].stControl.bInterlockBwd AND NOT gvl.astAxes[2].stControl.bInterlockFwd;

// NETWORK 6
main.stHWstatusY.bManualInterlockOverride := main.stHWControlY.bManualInterlockOverride;

// NETWORK 7
main.stHWstatusY.bSumBwdILOK := gvl.astAxes[2].stStatus.bBwEnabled AND NOT gvl.astAxes[2].stControl.bInterlockBwd;

// NETWORK 8
main.stHWstatusY.bSumFwdILOK := gvl.astAxes[2].stStatus.bFwEnabled AND NOT gvl.astAxes[2].stControl.bInterlockFwd;

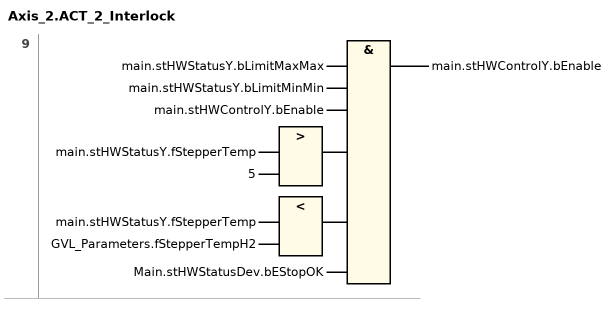
// NETWORK 9
main.stHWControlY.bEnable := main.stHWStatusY.bLimitMaxMax AND main.stHWStatusY.bLimitMinMin AND main.stHWControlY.bEnable AND main.stHWStatusY.fStepperTemp > 5 AND main.stHWStatusY.fStepperTemp < GVL_Parameters.fStepperTempH2 AND Main.stHWStatusDev.bEStopOK;
END_ACTION

END_PROGRAM

// ---- POUs/Application_Specific/Axes/Axis_3.TcPOU
PROGRAM Axis_3
VAR
	bLimitPowerAxis3 AT %Q*: BOOL := TRUE;
	temp: BOOL;
END_VAR
VAR // added by the converter: edge detectors and wires of the graphical bodies
    _w1, _w2 : BOOL;
END_VAR

//Initial parameters of an Axis
IF _TaskInfo[fbGetCurTaskIndex.index].FirstCycle THEN
    //Initial default values:
    GVL.astAxes[3].stConfig.eHomeSeq := 1;
    GVL.astAxes[3].stConfig.fHomePosition := 0.0;
    GVL.astAxes[3].stConfig.fHomeFinishDistance := 0;
END_IF

ACT_3_Interlock();

main.stHWStatusZ.bBrakeReleased:=FALSE;  // Not used
main.stHWControlZ.bBrakeReleaseCmd:=FALSE; // Not used

// Enable Cmd from GUI
GVL.astAxes[3].stControl.bEnable:=main.stHWControlZ.bEnable;
main.stHWStatusZ.bEnabled:=GVL.astAxes[3].stStatus.bEnabled;

// Trigger Abs movement from GUI
IF main.stHWControlZ.bExecuteAbsPos  AND NOT GVL.astAxes[3].stStatus.bBusy THEN
  GVL.astAxes[3].stControl.eCommand:=E_MotionFunctions.eMoveAbsolute;
  GVL.astAxes[3].stControl.bExecute:=TRUE;
  main.stHWControlZ.bExecuteAbsPos:=FALSE;
END_IF

// Trigger Const Velo movement from GUI
IF main.stHWControlZ.bExecuteConstVelo AND NOT GVL.astAxes[3].stStatus.bBusy THEN
  GVL.astAxes[3].stControl.eCommand:=E_MotionFunctions.eMoveVelocity;
  GVL.astAxes[3].stControl.bExecute:=TRUE;
  main.stHWControlZ.bExecuteConstVelo:=FALSE;
END_IF

// Trigger Home vs LimitFwd (should be valid for all axes) from GUI
IF main.stHWControlZ.bExecuteHome  AND NOT GVL.astAxes[3].stStatus.bBusy THEN
  GVL.astAxes[3].stConfig.fHomePosition:=GVL_Parameters.fZHomePosition;
  GVL.astAxes[3].stConfig.fHomingVelFromCam:=GVL_Parameters.fZHomeVelOffCam;
  GVL.astAxes[3].stConfig.fHomingVelToCam:=GVL_Parameters.fZHomeVelToCam;
  GVL.astAxes[3].stControl.eCommand:=E_MotionFunctions.eHome;
  GVL.astAxes[3].stConfig.eHomeSeq:=E_HomingRoutines.eHomeToLimit_Fwd;
  GVL.astAxes[3].stControl.bExecute:=TRUE;
  main.stHWControlZ.bExecuteHome:=FALSE;
END_IF

//Stop Motion from GUI
IF main.stHWControlZ.bExecuteStop THEN
  GVL.astAxes[3].stControl.bStop := NOT(GVL.astAxes[3].stControl.bStop);
  GVL.astAxes[3].stControl.bExecute:=FALSE;
  main.stHWControlZ.bExecuteStop:=FALSE;
END_IF

main.stHWStatusZ.bBusy:=GVL.astAxes[3].stStatus.bBusy;
GVL.astAxes[3].stControl.bReset:=main.stHWControlZ.bExecuteReset;
main.stHWControlZ.bExecuteReset:=FALSE;
main.stHWStatusZ.bHomed:=GVL.astAxes[3].stStatus.bHomed;
main.stHWStatusZ.bHomingCmdActive:=GVL.astAxes[3].stControl.eCommand=E_MotionFunctions.eHome AND 
                                   GVL.astAxes[3].stConfig.eHomeSeq=E_HomingRoutines.eHomeToLimit_Fwd;

// Hard code velocities and acc/dec
GVL.astAxes[3].stControl.fAcceleration:=GVL_Parameters.fZStepperTargetAcc;
GVL.astAxes[3].stControl.fDeceleration:=GVL_Parameters.fZStepperTargetAcc;
GVL.astAxes[3].stControl.fVelocity:=GVL_Parameters.fZStepperTargetVelo;

// reverse velo if dir is BWD
IF GVL.astAxes[3].stControl.eCommand=E_MotionFunctions.eMoveVelocity AND NOT main.stHWControlZ.bJogDirFwd  THEN
	GVL.astAxes[3].stControl.fVelocity:=-GVL_Parameters.fZStepperTargetVelo;
END_IF

// Check position is inside limits (and homed)
IF main.stHWStatusZ.bParkingRangeEnabled THEN 
  main.stHWStatusZ.bLoLoAlm:=gvl.astAxes[3].stStatus.fActPosition < GVL_Parameters.fZRangeParkL2 OR NOT main.stHWStatusZ.bHomed;
  main.stHWStatusZ.bLoAlm:=gvl.astAxes[3].stStatus.fActPosition < GVL_Parameters.fZRangeParkL1 OR NOT main.stHWStatusZ.bHomed;;
ELSE
  main.stHWStatusZ.bLoLoAlm:=gvl.astAxes[3].stStatus.fActPosition < GVL_Parameters.fZRangeL2 OR NOT main.stHWStatusZ.bHomed;;
  main.stHWStatusZ.bLoAlm:=gvl.astAxes[3].stStatus.fActPosition < GVL_Parameters.fZRangeL1 OR NOT main.stHWStatusZ.bHomed;;		
END_IF

main.stHWStatusZ.bHiAlm:=gvl.astAxes[3].stStatus.fActPosition > GVL_Parameters.fZRangeH1 OR NOT main.stHWStatusZ.bHomed;;
main.stHWStatusZ.bhiHiAlm:=gvl.astAxes[3].stStatus.fActPosition > GVL_Parameters.fZRangeH2 OR NOT main.stHWStatusZ.bHomed;;

ACTION ACT_3_Interlock:
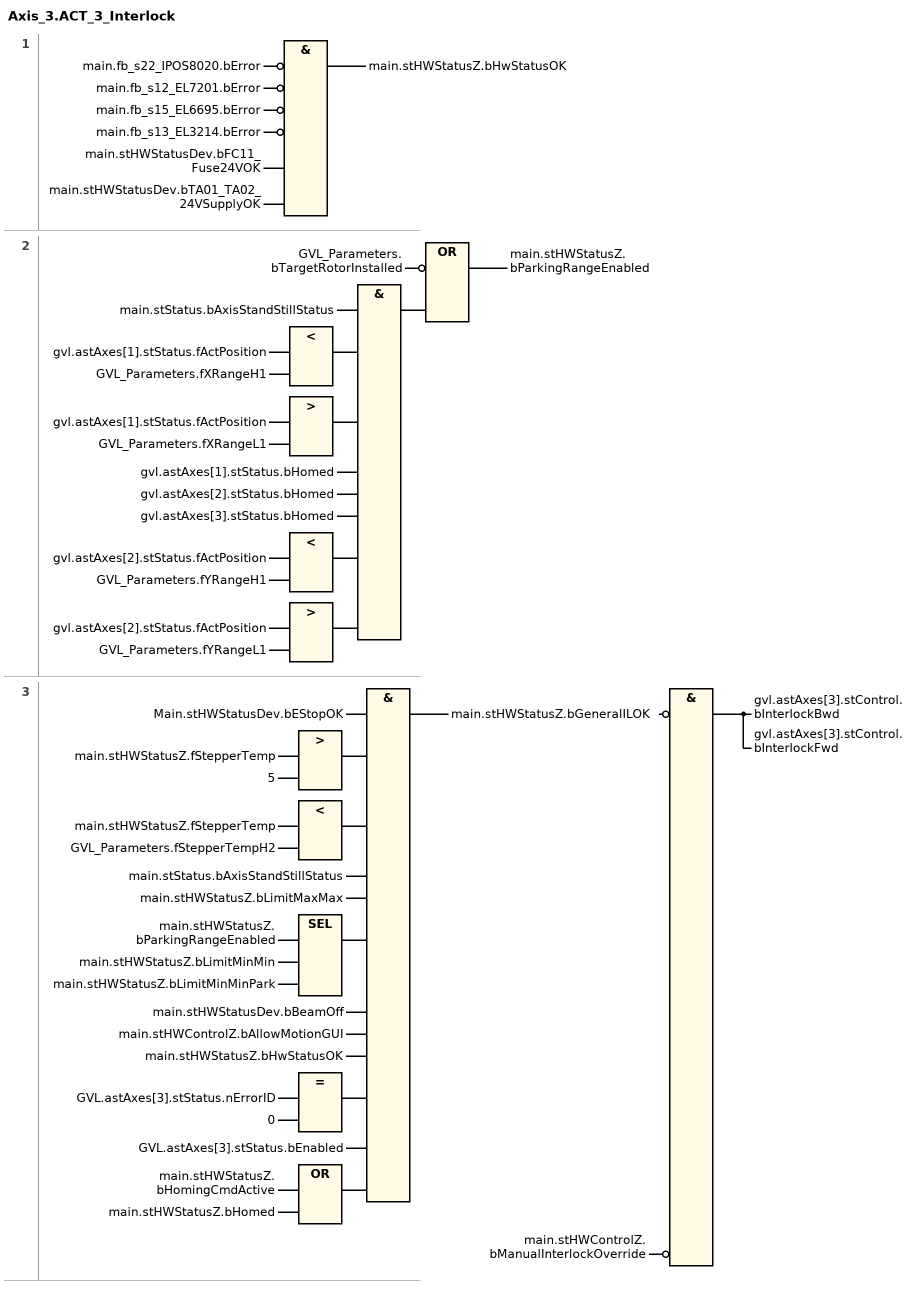
// NETWORK 1
main.stHWStatusZ.bHwStatusOK := NOT main.fb_s22_IPOS8020.bError AND NOT main.fb_s12_EL7201.bError AND NOT main.fb_s15_EL6695.bError AND NOT main.fb_s13_EL3214.bError AND main.stHWStatusDev.bFC11_Fuse24VOK AND main.stHWStatusDev.bTA01_TA02_24VSupplyOK;

// NETWORK 2
main.stHWStatusZ.bParkingRangeEnabled := NOT GVL_Parameters.bTargetRotorInstalled OR main.stStatus.bAxisStandStillStatus AND gvl.astAxes[1].stStatus.fActPosition < GVL_Parameters.fXRangeH1 AND gvl.astAxes[1].stStatus.fActPosition > GVL_Parameters.fXRangeL1 AND gvl.astAxes[1].stStatus.bHomed AND gvl.astAxes[2].stStatus.bHomed AND gvl.astAxes[3].stStatus.bHomed AND gvl.astAxes[2].stStatus.fActPosition < GVL_Parameters.fYRangeH1 AND gvl.astAxes[2].stStatus.fActPosition > GVL_Parameters.fYRangeL1;

// NETWORK 3
_w1 := Main.stHWStatusDev.bEStopOK AND main.stHWStatusZ.fStepperTemp > 5 AND main.stHWStatusZ.fStepperTemp < GVL_Parameters.fStepperTempH2 AND main.stStatus.bAxisStandStillStatus AND main.stHWStatusZ.bLimitMaxMax AND SEL(main.stHWStatusZ.bParkingRangeEnabled, main.stHWStatusZ.bLimitMinMin, main.stHWStatusZ.bLimitMinMinPark) AND main.stHWStatusDev.bBeamOff AND main.stHWControlZ.bAllowMotionGUI AND main.stHWStatusZ.bHwStatusOK AND GVL.astAxes[3].stStatus.nErrorID = 0 AND GVL.astAxes[3].stStatus.bEnabled AND (main.stHWStatusZ.bHomingCmdActive OR main.stHWStatusZ.bHomed);
main.stHWStatusZ.bGeneralILOK := _w1;
_w2 := NOT _w1 AND NOT main.stHWControlZ.bManualInterlockOverride;
gvl.astAxes[3].stControl.bInterlockBwd := _w2;
gvl.astAxes[3].stControl.bInterlockFwd := _w2;

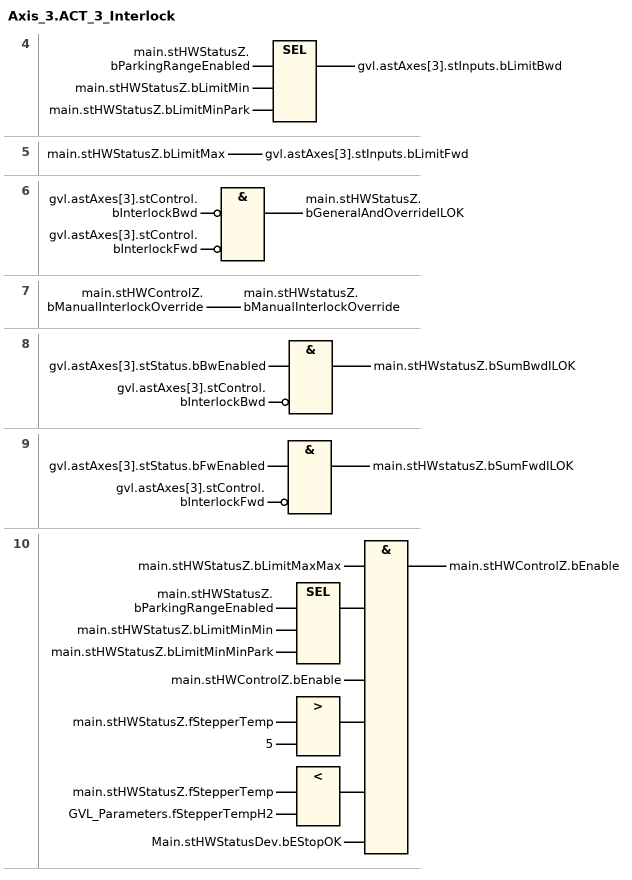
// NETWORK 4
gvl.astAxes[3].stInputs.bLimitBwd := SEL(main.stHWStatusZ.bParkingRangeEnabled, main.stHWStatusZ.bLimitMin, main.stHWStatusZ.bLimitMinPark);

// NETWORK 5
gvl.astAxes[3].stInputs.bLimitFwd := main.stHWStatusZ.bLimitMax;

// NETWORK 6
main.stHWStatusZ.bGeneralAndOverrideILOK := NOT gvl.astAxes[3].stControl.bInterlockBwd AND NOT gvl.astAxes[3].stControl.bInterlockFwd;

// NETWORK 7
main.stHWstatusZ.bManualInterlockOverride := main.stHWControlZ.bManualInterlockOverride;

// NETWORK 8
main.stHWstatusZ.bSumBwdILOK := gvl.astAxes[3].stStatus.bBwEnabled AND NOT gvl.astAxes[3].stControl.bInterlockBwd;

// NETWORK 9
main.stHWstatusZ.bSumFwdILOK := gvl.astAxes[3].stStatus.bFwEnabled AND NOT gvl.astAxes[3].stControl.bInterlockFwd;

// NETWORK 10
main.stHWControlZ.bEnable := main.stHWStatusZ.bLimitMaxMax AND SEL(main.stHWStatusZ.bParkingRangeEnabled, main.stHWStatusZ.bLimitMinMin, main.stHWStatusZ.bLimitMinMinPark) AND main.stHWControlZ.bEnable AND main.stHWStatusZ.fStepperTemp > 5 AND main.stHWStatusZ.fStepperTemp < GVL_Parameters.fStepperTempH2 AND Main.stHWStatusDev.bEStopOK;
END_ACTION

END_PROGRAM

// ---- POUs/Application_Specific/Applications/Application_Template.TcPOU
PROGRAM Application_Template
VAR
//Define all necessary variables for your application
END_VAR

//Program any specific code or safety code for an specific application when it involves multiple axes
//Eg. Collision avoidance, interlocks, sequencing, etc.

END_PROGRAM

// ---- POUs/Application_Specific/Axes/Axis_Template.TcPOU
PROGRAM Axis_Template
VAR

END_VAR

//Initial parameters of an Axis
(*IF _TaskInfo[fbGetCurTaskIndex.index].FirstCycle THEN
    //Initial default values:
    GVL.astAxes[1].stControl.fVelocity := GVL.astAxes[1].stConfig.fVelocityDefaultSlow;
    GVL.astAxes[1].stConfig.eHomeSeq := 0;
    GVL.astAxes[1].stConfig.fHomePosition := 0.0;
    GVL.astAxes[1].stConfig.fHomeFinishDistance := 0.0;
END_IF*)

//Define ACTIONS() or write exclusive code for an specific axis.
//Eg. Stop when temperature reaches certain values, reduce speed if  a signal is activated, etc.

END_PROGRAM

// ---- POUs/Common/ChangeConfig/FB_ReadFloatParameter.TcPOU
FUNCTION_BLOCK FB_ReadFloatParameter
VAR_INPUT
    bExecute: BOOL;
    ///16#4000=Axisdata, 16#5000=Encoderdata, 16#6000=Controldata, 16#7000=Drivedata
    nDeviceGroup: UDINT;
    nIndexOffset: UDINT;
END_VAR
VAR_OUTPUT
    nData: LREAL;
    bBusy: BOOL;
    bDone: BOOL;
    bError: BOOL;
    nErrorId: UDINT;
END_VAR
VAR_IN_OUT
    Axis: AXIS_REF;
END_VAR
VAR
    nState: UINT;
    fbADSREAD: ADSREAD;
END_VAR

(*Sequence to read parameter in Nc*)
CASE nState OF
0:  (*Start sequence. Wait until bExecute is TRUE*)
    IF bExecute THEN
        bBusy:=TRUE;
        bError:=FALSE;
        nErrorId:=0;
        nState:=10;
    END_IF

10: (*Read parameter in Nc*)
    fbADSREAD(
        PORT:=500,
        IDXGRP:=nDeviceGroup+Axis.NcToPlc.AxisId,
        IDXOFFS:=nIndexOffset,
        LEN:=SIZEOF(nData),
        DESTADDR:=ADR(nData),
        READ:=TRUE);

    (*Wait until it's done or if an error occurs*)
    IF NOT fbADSREAD.ERR THEN
        IF NOT fbADSREAD.BUSY THEN
            fbADSREAD(READ:=FALSE);
            nState:=20;
        END_IF
    ELSE
        nErrorId:=fbADSREAD.ERRID;
        nState:=999;
    END_IF

20: (*Sequense is done. Waits until bExecute is FALSE*)
    bBusy:=FALSE;
    bDone:=TRUE;
    IF NOT bExecute THEN
        bDone:=FALSE;
        nState:=0;
    END_IF

999: (*Error in sequence*)
    bError:=TRUE;
    bBusy:=FALSE;
    bDone:=FALSE;
    fbADSREAD(READ:=FALSE);
    IF NOT bExecute THEN
        nState:=0;
    END_IF

END_CASE

END_FUNCTION_BLOCK

// ---- POUs/Common/ChangeConfig/FB_ReadParameterInNc_v1_00.TcPOU
///#########################################################
///Function block to read parameter in Nc.
///
/// Library:
/// Tc2_MC2.lib
/// Tc2_System.lib
///
/// Global Variables:
///
/// Data types:
///
/// External functions:
///
/// History:
/// 2014-02-05  v1.00   NB  Release code.
///
/// Known bugs:
///
///
///
///###########################################################
FUNCTION_BLOCK FB_ReadParameterInNc_v1_00
VAR_INPUT
    bExecute: BOOL;
    ///16#4000=Axisdata, 16#5000=Encoderdata, 16#6000=Controldata, 16#7000=Drivedata
    nDeviceGroup: UDINT;
    nIndexOffset: UDINT;
END_VAR
VAR_OUTPUT
    nData: DWORD;
    bBusy: BOOL;
    bDone: BOOL;
    bError: BOOL;
    nErrorId: UDINT;
END_VAR
VAR_IN_OUT
    Axis: AXIS_REF;
END_VAR
VAR
    nState: UINT;
    fbADSREAD: ADSREAD;
END_VAR

(*Sequence to read parameter in Nc*)
CASE nState OF
0:  (*Start sequence. Wait until bExecute is TRUE*)
    IF bExecute THEN
        bBusy:=TRUE;
        bError:=FALSE;
        nErrorId:=0;
        nState:=10;
    END_IF

10: (*Read parameter in Nc*)
    fbADSREAD(
        PORT:=500,
        IDXGRP:=nDeviceGroup+Axis.NcToPlc.AxisId,
        IDXOFFS:=nIndexOffset,
        LEN:=SIZEOF(nData),
        DESTADDR:=ADR(nData),
        READ:=TRUE);

    (*Wait until it's done or if an error occurs*)
    IF NOT fbADSREAD.ERR THEN
        IF NOT fbADSREAD.BUSY THEN
            fbADSREAD(READ:=FALSE);
            nState:=20;
        END_IF
    ELSE
        nErrorId:=fbADSREAD.ERRID;
        nState:=999;
    END_IF

20: (*Sequense is done. Waits until bExecute is FALSE*)
    bBusy:=FALSE;
    bDone:=TRUE;
    IF NOT bExecute THEN
        bDone:=FALSE;
        nState:=0;
    END_IF

999: (*Error in sequence*)
    bError:=TRUE;
    bBusy:=FALSE;
    bDone:=FALSE;
    fbADSREAD(READ:=FALSE);
    IF NOT bExecute THEN
        nState:=0;
    END_IF

END_CASE

END_FUNCTION_BLOCK

// ---- POUs/Common/ChangeConfig/FB_WriteFloatParameter.TcPOU
///#########################################################
///Function block to write parameter in Nc.
///
/// Library:
/// Tc2_MC2.lib
/// Tc2_System.lib
///
/// Global Variables:
///
/// Data types:
///
/// External functions:
///
/// History:
/// 2014-02-05  v1.00   NB  Release code.
///
/// Known bugs:
///
///
///
///###########################################################
FUNCTION_BLOCK FB_WriteFloatParameter
VAR_INPUT
    bExecute: BOOL;
    ///16#4000=Axisdata, 16#5000=Encoderdata, 16#6000=Controldata, 16#7000=Drivedata
    nDeviceGroup: UDINT;
    nIndexOffset: UDINT;
    nData: LREAL;
END_VAR
VAR_OUTPUT
    bBusy: BOOL;
    bDone: BOOL;
    bError: BOOL;
    nErrorId: UDINT;
END_VAR
VAR_IN_OUT
    Axis: AXIS_REF;
END_VAR
VAR
    nState: UINT;
    fbADSWRITE: ADSWRITE;
END_VAR

(*Sequence to write parameter in Nc*)
CASE nState OF
0:  (*Start sequence. Wait until bExecute is TRUE*)
    IF bExecute THEN
        bBusy:=TRUE;
        bError:=FALSE;
        nErrorId:=0;
        nState:=10;
    END_IF

10: (*Write parameter in Nc*)
    fbADSWRITE(
        PORT:=500,
        IDXGRP:=nDeviceGroup+Axis.NcToPlc.AxisId,
        IDXOFFS:=nIndexOffset,
        LEN:=SIZEOF(nData),
        SRCADDR:=ADR(nData),
        WRITE:=TRUE);

    (*Wait until it's done or if an error occurs*)
    IF NOT fbADSWRITE.ERR THEN
        IF NOT fbADSWRITE.BUSY THEN
            fbADSWRITE(WRITE:=FALSE);
            nState:=20;
        END_IF
    ELSE
        nErrorId:=fbADSWRITE.ERRID;
        nState:=999;
    END_IF

20: (*Sequense is done. Waits until bExecute is FALSE*)
    bBusy:=FALSE;
    bDone:=TRUE;
    IF NOT bExecute THEN
        bDone:=FALSE;
        nState:=0;
    END_IF

999: (*Error in sequence*)
    bError:=TRUE;
    bBusy:=FALSE;
    bDone:=FALSE;
    fbADSWRITE(WRITE:=FALSE);
    IF NOT bExecute THEN
        nState:=0;
    END_IF

END_CASE

END_FUNCTION_BLOCK

// ---- POUs/Common/ChangeConfig/FB_WriteParameterInNc_v1_00.TcPOU
///#########################################################
///Function block to write parameter in Nc.
///
/// Library:
/// Tc2_MC2.lib
/// Tc2_System.lib
///
/// Global Variables:
///
/// Data types:
///
/// External functions:
///
/// History:
/// 2014-02-05  v1.00   NB  Release code.
///
/// Known bugs:
///
///
///
///###########################################################
FUNCTION_BLOCK FB_WriteParameterInNc_v1_00
VAR_INPUT
    bExecute: BOOL;
    ///16#4000=Axisdata, 16#5000=Encoderdata, 16#6000=Controldata, 16#7000=Drivedata
    nDeviceGroup: UDINT;
    nIndexOffset: UDINT;
    nData: DWORD;
END_VAR
VAR_OUTPUT
    bBusy: BOOL;
    bDone: BOOL;
    bError: BOOL;
    nErrorId: UDINT;
END_VAR
VAR_IN_OUT
    Axis: AXIS_REF;
END_VAR
VAR
    nState: UINT;
    fbADSWRITE: ADSWRITE;
END_VAR

(*Sequence to write parameter in Nc*)
CASE nState OF
0:  (*Start sequence. Wait until bExecute is TRUE*)
    IF bExecute THEN
        bBusy:=TRUE;
        bError:=FALSE;
        nErrorId:=0;
        nState:=10;
    END_IF

10: (*Write parameter in Nc*)
    fbADSWRITE(
        PORT:=500,
        IDXGRP:=nDeviceGroup+Axis.NcToPlc.AxisId,
        IDXOFFS:=nIndexOffset,
        LEN:=SIZEOF(nData),
        SRCADDR:=ADR(nData),
        WRITE:=TRUE);

    (*Wait until it's done or if an error occurs*)
    IF NOT fbADSWRITE.ERR THEN
        IF NOT fbADSWRITE.BUSY THEN
            fbADSWRITE(WRITE:=FALSE);
            nState:=20;
        END_IF
    ELSE
        nErrorId:=fbADSWRITE.ERRID;
        nState:=999;
    END_IF

20: (*Sequense is done. Waits until bExecute is FALSE*)
    bBusy:=FALSE;
    bDone:=TRUE;
    IF NOT bExecute THEN
        bDone:=FALSE;
        nState:=0;
    END_IF

999: (*Error in sequence*)
    bError:=TRUE;
    bBusy:=FALSE;
    bDone:=FALSE;
    fbADSWRITE(WRITE:=FALSE);
    IF NOT bExecute THEN
        nState:=0;
    END_IF

END_CASE

END_FUNCTION_BLOCK

// ---- POUs/Common/ErrorHandling/FB_NC_Error.TcPOU
FUNCTION_BLOCK FB_NC_Error

VAR_INPUT
    En              : BOOL;
    nNC_ErrorID     : UDINT;
    nNC_AxisID      : UDINT;
    ErrorSystem     : POINTER TO ST_ErrorSystem;
END_VAR

VAR_OUTPUT
    EnO         : BOOL;
    bError      : BOOL;
END_VAR

VAR
    NCError             : FB_GenericError;
END_VAR

(*
* ================================================================================
*                                   DESCRIPTION
* ================================================================================
* This Function Block connects FB_DriveVirtual's error output to the Error System.
* Link the corresponding outputs of FB_DriveVirtual to the inputs of this FB.
* ================================================================================
*)

IF En THEN
    EnO := En;

    IF nNC_ErrorID <> 0 THEN
        NCError.sErrorMessage   := 'Axis ';
        NCError.sErrorMessage   := CONCAT (NCError.sErrorMessage, UDINT_TO_STRING(nNC_AxisID));
        NCError.sErrorMessage   := CONCAT (NCError.sErrorMessage, ' is in error state. NC error ID (Hex): 0x');
        NCError.sErrorMessage   := CONCAT (NCError.sErrorMessage, DWORD_TO_HEXSTR(nNC_ErrorID,4,FALSE));
        NCError.ErrorPriority   := 6;
        NCError.bError          := TRUE;
    ELSE
        NCError.sErrorMessage   := '';
        NCError.bError          := FALSE;
        NCError.ErrorPriority   := 0;
    END_IF

END_IF

NCError (
    En                  := TRUE,
    bError              := ,
    sErrorMessage       := ,
    ErrorPriority       := ,
    iTerminal_ID        := ,
    pErrorSystem        := ErrorSystem,
    EnO     => ,
);


(*
        NCError.sErrorMessage := CONCAT (NCError.sErrorMessage, ': ');
        CASE nNC_ErrorID OF
            //General NC Errors
            16#4000 :   NCError.sErrorMessage := CONCAT (NCError.sErrorMessage,     'Internal Error; ');
            16#4001 :   NCError.sErrorMessage := CONCAT (NCError.sErrorMessage,     'Memory Error; ');
            16#4002 :   NCError.sErrorMessage := CONCAT (NCError.sErrorMessage,     'NC retain data error (persistent data); ');
            16#4010 :   NCError.sErrorMessage := CONCAT (NCError.sErrorMessage,     'Channel identifier not allowed; ');
            16#4011 :   NCError.sErrorMessage := CONCAT (NCError.sErrorMessage,     'Group identifier not allowed; ');
            16#4012 :   NCError.sErrorMessage := CONCAT (NCError.sErrorMessage,     'Axis identifier not allowed; ');
            16#4013 :   NCError.sErrorMessage := CONCAT (NCError.sErrorMessage,     'Encoder identifier not allowed; ');
            16#4014 :   NCError.sErrorMessage := CONCAT (NCError.sErrorMessage,     'Controller identifier not allowed; ');
            16#4015 :   NCError.sErrorMessage := CONCAT (NCError.sErrorMessage,     'Drive identifier not allowed; ');
            16#4016 :   NCError.sErrorMessage := CONCAT (NCError.sErrorMessage,     'Table identifier not allowed; ');
            16#4020 :   NCError.sErrorMessage := CONCAT (NCError.sErrorMessage,     'No process image; ');
            16#4021 :   NCError.sErrorMessage := CONCAT (NCError.sErrorMessage,     'No process image; ');
            16#4022 :   NCError.sErrorMessage := CONCAT (NCError.sErrorMessage,     'No process image; ');
            16#4023 :   NCError.sErrorMessage := CONCAT (NCError.sErrorMessage,     'No process image; ');
            16#4024 :   NCError.sErrorMessage := CONCAT (NCError.sErrorMessage,     'No process image; ');
            16#4025 :   NCError.sErrorMessage := CONCAT (NCError.sErrorMessage,     'No process image; ');
            16#4030 :   NCError.sErrorMessage := CONCAT (NCError.sErrorMessage,     'Coupling type not allowed; ');
            16#4031 :   NCError.sErrorMessage := CONCAT (NCError.sErrorMessage,     'Axis type not allowed; ');
            16#4040 :   NCError.sErrorMessage := CONCAT (NCError.sErrorMessage,     'Axis is incompatible; ');
            16#4050 :   NCError.sErrorMessage := CONCAT (NCError.sErrorMessage,     'Channel not ready for operation; ');
            16#4051 :   NCError.sErrorMessage := CONCAT (NCError.sErrorMessage,     'Group not ready for operation; ');
            16#4052 :   NCError.sErrorMessage := CONCAT (NCError.sErrorMessage,     'Axis not ready for operation; ');
            16#4060 :   NCError.sErrorMessage := CONCAT (NCError.sErrorMessage,     'Channel exists; ');
            16#4061 :   NCError.sErrorMessage := CONCAT (NCError.sErrorMessage,     'Group exists; ');
            16#4062 :   NCError.sErrorMessage := CONCAT (NCError.sErrorMessage,     'Axis exists; ');
            16#4063 :   NCError.sErrorMessage := CONCAT (NCError.sErrorMessage,     'Table exists; ');
            16#4070 :   NCError.sErrorMessage := CONCAT (NCError.sErrorMessage,     'Axis index not allowed; ');
            16#4071 :   NCError.sErrorMessage := CONCAT (NCError.sErrorMessage,     'Axis index not allowed; ');

            //Channel Errors
            16#4101 :   NCError.sErrorMessage := CONCAT (NCError.sErrorMessage,     'Group index not allowed; ');
            16#4102 :   NCError.sErrorMessage := CONCAT (NCError.sErrorMessage,     'Null pointer; ');
            16#4103 :   NCError.sErrorMessage := CONCAT (NCError.sErrorMessage,     'No process image; ');
            16#4104 :   NCError.sErrorMessage := CONCAT (NCError.sErrorMessage,     'M-function index not allowed; ');
            16#4105 :   NCError.sErrorMessage := CONCAT (NCError.sErrorMessage,     'No memmory; ');
            16#4106 :   NCError.sErrorMessage := CONCAT (NCError.sErrorMessage,     'Not ready; ');
            16#4107 :   NCError.sErrorMessage := CONCAT (NCError.sErrorMessage,     'Function/command not supported; ');
            16#4108 :   NCError.sErrorMessage := CONCAT (NCError.sErrorMessage,     'Invalid parameter while starting; ');
            16#4109 :   NCError.sErrorMessage := CONCAT (NCError.sErrorMessage,     'Channel function/command not executable; ');
            16#410A :   NCError.sErrorMessage := CONCAT (NCError.sErrorMessage,     'ItpGoAhead not executable; ');
            16#4110 :   NCError.sErrorMessage := CONCAT (NCError.sErrorMessage,     'Error opening a file; ');
            16#4111 :   NCError.sErrorMessage := CONCAT (NCError.sErrorMessage,     'Syntax error during loading; ');
            16#4112 :   NCError.sErrorMessage := CONCAT (NCError.sErrorMessage,     'Syntax error  during interpretation; ');
            16#4113 :   NCError.sErrorMessage := CONCAT (NCError.sErrorMessage,     'Missing subroutine; ');
            16#4114 :   NCError.sErrorMessage := CONCAT (NCError.sErrorMessage,     'Loading buffer of interpreter is too small; ');
            16#4117 :   NCError.sErrorMessage := CONCAT (NCError.sErrorMessage,     'Subroutine incomplete; ');
            16#4118 :   NCError.sErrorMessage := CONCAT (NCError.sErrorMessage,     'Error while loading the NC program; ');
            16#4119 :   NCError.sErrorMessage := CONCAT (NCError.sErrorMessage,     'Error while loading the NC program; ');
            16#4120 :   NCError.sErrorMessage := CONCAT (NCError.sErrorMessage,     'Devide by zero; ');
            16#4121 :   NCError.sErrorMessage := CONCAT (NCError.sErrorMessage,     'Invalide circle parameterization; ');
            16#4122 :   NCError.sErrorMessage := CONCAT (NCError.sErrorMessage,     'Invalid FPU-Operation; ');
            16#4130 :   NCError.sErrorMessage := CONCAT (NCError.sErrorMessage,     'Stack overflow: subroutines; ');
            16#4131 :   NCError.sErrorMessage := CONCAT (NCError.sErrorMessage,     'Stack underflow: subroutines; ');
            16#4132 :   NCError.sErrorMessage := CONCAT (NCError.sErrorMessage,     'Stack overflow: arithmetic unit; ');
            16#4133 :   NCError.sErrorMessage := CONCAT (NCError.sErrorMessage,     'Stack underflow: arithmetic unit; ');
            16#4140 :   NCError.sErrorMessage := CONCAT (NCError.sErrorMessage,     'Register index not allowed; ');
            16#4141 :   NCError.sErrorMessage := CONCAT (NCError.sErrorMessage,     'Unaccaptable G-function index; ');
            16#4142 :   NCError.sErrorMessage := CONCAT (NCError.sErrorMessage,     'Unaccaptable M-function index; ');
            16#4143 :   NCError.sErrorMessage := CONCAT (NCError.sErrorMessage,     'Unacceptable extended address; ');
            16#4144 :   NCError.sErrorMessage := CONCAT (NCError.sErrorMessage,     'Unaccaptable index of internal H-function; ');
            16#4145 :   NCError.sErrorMessage := CONCAT (NCError.sErrorMessage,     'Machine data value unacceptable; ');
            16#4150 :   NCError.sErrorMessage := CONCAT (NCError.sErrorMessage,     'Cannot change tool params here; ');
            16#4151 :   NCError.sErrorMessage := CONCAT (NCError.sErrorMessage,     'Cannoot calculate tool compensation; ');
            16#4152 :   NCError.sErrorMessage := CONCAT (NCError.sErrorMessage,     'Tool compensation; ');
            16#4153 :   NCError.sErrorMessage := CONCAT (NCError.sErrorMessage,     'Tool compensation; ');
            16#4153 :   NCError.sErrorMessage := CONCAT (NCError.sErrorMessage,     'Tool compensation; ');


        END_CASE
*)

END_FUNCTION_BLOCK

// ---- POUs/Common/Hardware/EtherCAT_Terminals/Analog_Inputs/EL3174_0002.TcPOU
//EL3174-0002 | 4-channel analog input, -10/0...+10V, -20/0/+4...20mA, 16 bit, differential
FUNCTION_BLOCK EL3174_0002

VAR_INPUT
    En              : BOOL;
    iTerminal_ID    : INT;
    ErrorSystem     : POINTER TO ST_ErrorSystem;
END_VAR

VAR_OUTPUT
    EnO     : BOOL;
    bError  : BOOL;
END_VAR

VAR
    //Channels
    wCH1_Status     AT %I*  : WORD;
    wCH2_Status     AT %I*  : WORD;
    wCH3_Status     AT %I*  : WORD;
    wCH4_Status     AT %I*  : WORD;

    //Terminal status
    WcState_WcState AT %I*  : BOOL;
    InfoData_State  AT %I*  : UINT;

    //FB-s
    EL3174_0002_Error   : FB_TerminalError;
    CH1_Error           : FB_GenericError;
    CH2_Error           : FB_GenericError;
    CH3_Error           : FB_GenericError;
    CH4_Error           : FB_GenericError;
END_VAR

(*
* TODO: Test on hardware
*)
EnO := En;

IF En THEN
    //Channel #1 Status
    IF (wCh1_Status AND 16#2057) <> 0 THEN
        CH1_Error.sErrorMessage := 'EL3174-0002 Channel #1: ';
        IF wCH1_Status.0    THEN    CH1_Error.sErrorMessage := CONCAT(CH1_Error.sErrorMessage, 'Underrange; ');             IF CH1_Error.ErrorPriority > 100 OR CH1_Error.ErrorPriority = 0     THEN CH1_Error.ErrorPriority := 100;    END_IF      END_IF
        IF wCH1_Status.1    THEN    CH1_Error.sErrorMessage := CONCAT(CH1_Error.sErrorMessage, 'Overrange; ');              IF CH1_Error.ErrorPriority > 100 OR CH1_Error.ErrorPriority = 0     THEN CH1_Error.ErrorPriority := 100;    END_IF      END_IF
        IF wCh1_Status.2    THEN    CH1_Error.sErrorMessage := CONCAT(CH1_Error.sErrorMessage, 'Limit 1; ');                IF CH1_Error.ErrorPriority > 100 OR CH1_Error.ErrorPriority = 0     THEN CH1_Error.ErrorPriority := 100;    END_IF      END_IF
        IF wCh1_Status.4    THEN    CH1_Error.sErrorMessage := CONCAT(CH1_Error.sErrorMessage, 'Limit 2; ');                IF CH1_Error.ErrorPriority > 100 OR CH1_Error.ErrorPriority = 0     THEN CH1_Error.ErrorPriority := 100;    END_IF      END_IF
        IF wCh1_Status.6    THEN    CH1_Error.sErrorMessage := CONCAT(CH1_Error.sErrorMessage, 'Error; ');                  IF CH1_Error.ErrorPriority > 10  OR CH1_Error.ErrorPriority = 0     THEN CH1_Error.ErrorPriority := 10;     END_IF      END_IF
        IF wCh1_Status.13   THEN    CH1_Error.sErrorMessage := CONCAT(CH1_Error.sErrorMessage, 'Sync error; ');             IF CH1_Error.ErrorPriority > 10  OR CH1_Error.ErrorPriority = 0     THEN CH1_Error.ErrorPriority := 10;     END_IF      END_IF
        CH1_Error.bError := TRUE;
    ELSE
        CH1_Error.bError        := FALSE;
        CH1_Error.sErrorMessage := '';
    END_IF

    //Channel #2 Status
    IF (wCh2_Status AND 16#2057) <> 0 THEN
        CH2_Error.sErrorMessage := 'EL3174-0002 Channel #2: ';
        IF wCH2_Status.0    THEN    CH2_Error.sErrorMessage := CONCAT(CH2_Error.sErrorMessage, 'Underrange; ');             IF CH2_Error.ErrorPriority > 100 OR CH2_Error.ErrorPriority = 0     THEN CH2_Error.ErrorPriority := 100;    END_IF      END_IF
        IF wCH2_Status.1    THEN    CH2_Error.sErrorMessage := CONCAT(CH2_Error.sErrorMessage, 'Overrange; ');              IF CH2_Error.ErrorPriority > 100 OR CH2_Error.ErrorPriority = 0     THEN CH2_Error.ErrorPriority := 100;    END_IF      END_IF
        IF wCh2_Status.2    THEN    CH2_Error.sErrorMessage := CONCAT(CH2_Error.sErrorMessage, 'Limit 1; ');                IF CH2_Error.ErrorPriority > 100 OR CH2_Error.ErrorPriority = 0     THEN CH2_Error.ErrorPriority := 100;    END_IF      END_IF
        IF wCh2_Status.4    THEN    CH2_Error.sErrorMessage := CONCAT(CH2_Error.sErrorMessage, 'Limit 2; ');                IF CH2_Error.ErrorPriority > 100 OR CH2_Error.ErrorPriority = 0     THEN CH2_Error.ErrorPriority := 100;    END_IF      END_IF
        IF wCh2_Status.6    THEN    CH2_Error.sErrorMessage := CONCAT(CH2_Error.sErrorMessage, 'Error; ');                  IF CH2_Error.ErrorPriority > 10  OR CH2_Error.ErrorPriority = 0     THEN CH2_Error.ErrorPriority := 10;     END_IF      END_IF
        IF wCh2_Status.13   THEN    CH2_Error.sErrorMessage := CONCAT(CH2_Error.sErrorMessage, 'Sync error; ');             IF CH2_Error.ErrorPriority > 10  OR CH2_Error.ErrorPriority = 0     THEN CH2_Error.ErrorPriority := 10;     END_IF      END_IF
        CH2_Error.bError := TRUE;
    ELSE
        CH2_Error.bError        := FALSE;
        CH2_Error.sErrorMessage := '';
    END_IF

    //Channel #3 Status
    IF (wCh3_Status AND 16#2057) <> 0 THEN
        CH3_Error.sErrorMessage := 'EL3174-0002 Channel #3: ';
        IF wCH3_Status.0    THEN    CH3_Error.sErrorMessage := CONCAT(CH3_Error.sErrorMessage, 'Underrange; ');             IF CH3_Error.ErrorPriority > 100 OR CH3_Error.ErrorPriority = 0     THEN CH3_Error.ErrorPriority := 100;    END_IF      END_IF
        IF wCH3_Status.1    THEN    CH3_Error.sErrorMessage := CONCAT(CH3_Error.sErrorMessage, 'Overrange; ');              IF CH3_Error.ErrorPriority > 100 OR CH3_Error.ErrorPriority = 0     THEN CH3_Error.ErrorPriority := 100;    END_IF      END_IF
        IF wCh3_Status.2    THEN    CH3_Error.sErrorMessage := CONCAT(CH3_Error.sErrorMessage, 'Limit 1; ');                IF CH3_Error.ErrorPriority > 100 OR CH3_Error.ErrorPriority = 0     THEN CH3_Error.ErrorPriority := 100;    END_IF      END_IF
        IF wCh3_Status.4    THEN    CH3_Error.sErrorMessage := CONCAT(CH3_Error.sErrorMessage, 'Limit 2; ');                IF CH3_Error.ErrorPriority > 100 OR CH3_Error.ErrorPriority = 0     THEN CH3_Error.ErrorPriority := 100;    END_IF      END_IF
        IF wCh3_Status.6    THEN    CH3_Error.sErrorMessage := CONCAT(CH3_Error.sErrorMessage, 'Error; ');                  IF CH3_Error.ErrorPriority > 10  OR CH3_Error.ErrorPriority = 0     THEN CH3_Error.ErrorPriority := 10;     END_IF      END_IF
        IF wCh3_Status.13   THEN    CH3_Error.sErrorMessage := CONCAT(CH3_Error.sErrorMessage, 'Sync error; ');             IF CH3_Error.ErrorPriority > 10  OR CH3_Error.ErrorPriority = 0     THEN CH3_Error.ErrorPriority := 10;     END_IF      END_IF
        CH3_Error.bError := TRUE;
    ELSE
        CH3_Error.bError        := FALSE;
        CH3_Error.sErrorMessage := '';
    END_IF

    //Channel #4 Status
    IF (wCh4_Status AND 16#2057) <> 0 THEN
        CH4_Error.sErrorMessage := 'EL3174-0002 Channel #4: ';
        IF wCH4_Status.0    THEN    CH4_Error.sErrorMessage := CONCAT(CH4_Error.sErrorMessage, 'Underrange; ');             IF CH4_Error.ErrorPriority > 100 OR CH4_Error.ErrorPriority = 0     THEN CH4_Error.ErrorPriority := 100;    END_IF      END_IF
        IF wCH4_Status.1    THEN    CH4_Error.sErrorMessage := CONCAT(CH4_Error.sErrorMessage, 'Overrange; ');              IF CH4_Error.ErrorPriority > 100 OR CH4_Error.ErrorPriority = 0     THEN CH4_Error.ErrorPriority := 100;    END_IF      END_IF
        IF wCh4_Status.2    THEN    CH4_Error.sErrorMessage := CONCAT(CH4_Error.sErrorMessage, 'Limit 1; ');                IF CH4_Error.ErrorPriority > 100 OR CH4_Error.ErrorPriority = 0     THEN CH4_Error.ErrorPriority := 100;    END_IF      END_IF
        IF wCh4_Status.4    THEN    CH4_Error.sErrorMessage := CONCAT(CH4_Error.sErrorMessage, 'Limit 2; ');                IF CH4_Error.ErrorPriority > 100 OR CH4_Error.ErrorPriority = 0     THEN CH4_Error.ErrorPriority := 100;    END_IF      END_IF
        IF wCh4_Status.6    THEN    CH4_Error.sErrorMessage := CONCAT(CH4_Error.sErrorMessage, 'Error; ');                  IF CH4_Error.ErrorPriority > 10  OR CH4_Error.ErrorPriority = 0     THEN CH4_Error.ErrorPriority := 10;     END_IF      END_IF
        IF wCh4_Status.13   THEN    CH4_Error.sErrorMessage := CONCAT(CH4_Error.sErrorMessage, 'Sync error; ');             IF CH4_Error.ErrorPriority > 10  OR CH4_Error.ErrorPriority = 0     THEN CH4_Error.ErrorPriority := 10;     END_IF      END_IF
        CH4_Error.bError := TRUE;
    ELSE
        CH4_Error.bError        := FALSE;
        CH4_Error.sErrorMessage := '';
    END_IF

END_IF



//Error FB instance
EL3174_0002_Error(
    En                  := TRUE,
    iTerminal_ID        := iTerminal_ID,
    bWcState            := WcState_WcState,
    uiInfoData_State    := InfoData_State,
    pErrorSystem        := ErrorSystem,
    bError              => bError,
);

CH1_Error (
    En              := En,
    bError          := ,
    sErrorMessage   := ,
    ErrorPriority   := ,
    iTerminal_ID    := iTerminal_ID,
    pErrorSystem    := ErrorSystem,
    EnO             => ,
);

CH2_Error (
    En              := En,
    bError          := ,
    sErrorMessage   := ,
    ErrorPriority   := ,
    iTerminal_ID    := iTerminal_ID,
    pErrorSystem    := ErrorSystem,
    EnO             => ,
);

CH3_Error (
    En              := En,
    bError          := ,
    sErrorMessage   := ,
    ErrorPriority   := ,
    iTerminal_ID    := iTerminal_ID,
    pErrorSystem    := ErrorSystem,
    EnO             => ,
);

CH4_Error (
    En              := En,
    bError          := ,
    sErrorMessage   := ,
    ErrorPriority   := ,
    iTerminal_ID    := iTerminal_ID,
    pErrorSystem    := ErrorSystem,
    EnO             => ,
);

END_FUNCTION_BLOCK

// ---- POUs/Common/Hardware/EtherCAT_Terminals/Analog_Inputs/EL3255.TcPOU
//EL3255 | 5-channel potentiometer measurement with sensor supply
FUNCTION_BLOCK EL3255

VAR_INPUT
    En              : BOOL;
    iTerminal_ID    : INT;
    ErrorSystem     : POINTER TO ST_ErrorSystem;
END_VAR

VAR_OUTPUT
    EnO     : BOOL;
    bError  : BOOL;
END_VAR

VAR
    wCH1_Status     AT %I*  : WORD;
    wCH2_Status     AT %I*  : WORD;
    wCH3_Status     AT %I*  : WORD;
    wCH4_Status     AT %I*  : WORD;
    wCH5_Status     AT %I*  : WORD;
    WcState_WcState AT %I*  : BOOL;
    InfoData_State  AT %I*  : UINT;

    //FB-s
    EL3255_Error    : FB_TerminalError;
    CH1_Error       : FB_GenericError;
    CH2_Error       : FB_GenericError;
    CH3_Error       : FB_GenericError;
    CH4_Error       : FB_GenericError;
    CH5_Error       : FB_GenericError;
END_VAR

(*
* TODO: Test on hardware
*)
EnO:=En;

IF En THEN
    //Channel #1 Status
    IF (wCh1_Status AND 16#2057) <> 0 THEN
        CH1_Error.sErrorMessage := 'EL3255 Channel #1: ';
        IF wCH1_Status.0    THEN    CH1_Error.sErrorMessage := CONCAT(CH1_Error.sErrorMessage, 'Underrange; ');             IF CH1_Error.ErrorPriority > 100 OR CH1_Error.ErrorPriority = 0     THEN CH1_Error.ErrorPriority := 100;    END_IF      END_IF
        IF wCH1_Status.1    THEN    CH1_Error.sErrorMessage := CONCAT(CH1_Error.sErrorMessage, 'Overrange; ');              IF CH1_Error.ErrorPriority > 100 OR CH1_Error.ErrorPriority = 0     THEN CH1_Error.ErrorPriority := 100;    END_IF      END_IF
        IF wCh1_Status.2    THEN    CH1_Error.sErrorMessage := CONCAT(CH1_Error.sErrorMessage, 'Limit 1; ');                IF CH1_Error.ErrorPriority > 100 OR CH1_Error.ErrorPriority = 0     THEN CH1_Error.ErrorPriority := 100;    END_IF      END_IF
        IF wCh1_Status.4    THEN    CH1_Error.sErrorMessage := CONCAT(CH1_Error.sErrorMessage, 'Limit 2; ');                IF CH1_Error.ErrorPriority > 100 OR CH1_Error.ErrorPriority = 0     THEN CH1_Error.ErrorPriority := 100;    END_IF      END_IF
        IF wCh1_Status.6    THEN    CH1_Error.sErrorMessage := CONCAT(CH1_Error.sErrorMessage, 'Error; ');                  IF CH1_Error.ErrorPriority > 10  OR CH1_Error.ErrorPriority = 0     THEN CH1_Error.ErrorPriority := 10;     END_IF      END_IF
        IF wCh1_Status.13   THEN    CH1_Error.sErrorMessage := CONCAT(CH1_Error.sErrorMessage, 'Sync error; ');             IF CH1_Error.ErrorPriority > 10  OR CH1_Error.ErrorPriority = 0     THEN CH1_Error.ErrorPriority := 10;     END_IF      END_IF
        CH1_Error.bError := TRUE;
    ELSE
        CH1_Error.bError        := FALSE;
        CH1_Error.sErrorMessage := '';
    END_IF

    //Channel #2 Status
    IF (wCh2_Status AND 16#2057) <> 0 THEN
        CH2_Error.sErrorMessage := 'EL3255 Channel #2: ';
        IF wCH2_Status.0    THEN    CH2_Error.sErrorMessage := CONCAT(CH2_Error.sErrorMessage, 'Underrange; ');             IF CH2_Error.ErrorPriority > 100 OR CH2_Error.ErrorPriority = 0     THEN CH2_Error.ErrorPriority := 100;    END_IF      END_IF
        IF wCH2_Status.1    THEN    CH2_Error.sErrorMessage := CONCAT(CH2_Error.sErrorMessage, 'Overrange; ');              IF CH2_Error.ErrorPriority > 100 OR CH2_Error.ErrorPriority = 0     THEN CH2_Error.ErrorPriority := 100;    END_IF      END_IF
        IF wCh2_Status.2    THEN    CH2_Error.sErrorMessage := CONCAT(CH2_Error.sErrorMessage, 'Limit 1; ');                IF CH2_Error.ErrorPriority > 100 OR CH2_Error.ErrorPriority = 0     THEN CH2_Error.ErrorPriority := 100;    END_IF      END_IF
        IF wCh2_Status.4    THEN    CH2_Error.sErrorMessage := CONCAT(CH2_Error.sErrorMessage, 'Limit 2; ');                IF CH2_Error.ErrorPriority > 100 OR CH2_Error.ErrorPriority = 0     THEN CH2_Error.ErrorPriority := 100;    END_IF      END_IF
        IF wCh2_Status.6    THEN    CH2_Error.sErrorMessage := CONCAT(CH2_Error.sErrorMessage, 'Error; ');                  IF CH2_Error.ErrorPriority > 10  OR CH2_Error.ErrorPriority = 0     THEN CH2_Error.ErrorPriority := 10;     END_IF      END_IF
        IF wCh2_Status.13   THEN    CH2_Error.sErrorMessage := CONCAT(CH2_Error.sErrorMessage, 'Sync error; ');             IF CH2_Error.ErrorPriority > 10  OR CH2_Error.ErrorPriority = 0     THEN CH2_Error.ErrorPriority := 10;     END_IF      END_IF
        CH2_Error.bError := TRUE;
    ELSE
        CH2_Error.bError        := FALSE;
        CH2_Error.sErrorMessage := '';
    END_IF

    //Channel #3 Status
    IF (wCh3_Status AND 16#2057) <> 0 THEN
        CH3_Error.sErrorMessage := 'EL3255 Channel #3: ';
        IF wCH3_Status.0    THEN    CH3_Error.sErrorMessage := CONCAT(CH3_Error.sErrorMessage, 'Underrange; ');             IF CH3_Error.ErrorPriority > 100 OR CH3_Error.ErrorPriority = 0     THEN CH3_Error.ErrorPriority := 100;    END_IF      END_IF
        IF wCH3_Status.1    THEN    CH3_Error.sErrorMessage := CONCAT(CH3_Error.sErrorMessage, 'Overrange; ');              IF CH3_Error.ErrorPriority > 100 OR CH3_Error.ErrorPriority = 0     THEN CH3_Error.ErrorPriority := 100;    END_IF      END_IF
        IF wCh3_Status.2    THEN    CH3_Error.sErrorMessage := CONCAT(CH3_Error.sErrorMessage, 'Limit 1; ');                IF CH3_Error.ErrorPriority > 100 OR CH3_Error.ErrorPriority = 0     THEN CH3_Error.ErrorPriority := 100;    END_IF      END_IF
        IF wCh3_Status.4    THEN    CH3_Error.sErrorMessage := CONCAT(CH3_Error.sErrorMessage, 'Limit 2; ');                IF CH3_Error.ErrorPriority > 100 OR CH3_Error.ErrorPriority = 0     THEN CH3_Error.ErrorPriority := 100;    END_IF      END_IF
        IF wCh3_Status.6    THEN    CH3_Error.sErrorMessage := CONCAT(CH3_Error.sErrorMessage, 'Error; ');                  IF CH3_Error.ErrorPriority > 10  OR CH3_Error.ErrorPriority = 0     THEN CH3_Error.ErrorPriority := 10;     END_IF      END_IF
        IF wCh3_Status.13   THEN    CH3_Error.sErrorMessage := CONCAT(CH3_Error.sErrorMessage, 'Sync error; ');             IF CH3_Error.ErrorPriority > 10  OR CH3_Error.ErrorPriority = 0     THEN CH3_Error.ErrorPriority := 10;     END_IF      END_IF
        CH3_Error.bError := TRUE;
    ELSE
        CH3_Error.bError        := FALSE;
        CH3_Error.sErrorMessage := '';
    END_IF

    //Channel #4 Status
    IF (wCh4_Status AND 16#2057) <> 0 THEN
        CH4_Error.sErrorMessage := 'EL3255 Channel #4: ';
        IF wCH4_Status.0    THEN    CH4_Error.sErrorMessage := CONCAT(CH4_Error.sErrorMessage, 'Underrange; ');             IF CH4_Error.ErrorPriority > 100 OR CH4_Error.ErrorPriority = 0     THEN CH4_Error.ErrorPriority := 100;    END_IF      END_IF
        IF wCH4_Status.1    THEN    CH4_Error.sErrorMessage := CONCAT(CH4_Error.sErrorMessage, 'Overrange; ');              IF CH4_Error.ErrorPriority > 100 OR CH4_Error.ErrorPriority = 0     THEN CH4_Error.ErrorPriority := 100;    END_IF      END_IF
        IF wCh4_Status.2    THEN    CH4_Error.sErrorMessage := CONCAT(CH4_Error.sErrorMessage, 'Limit 1; ');                IF CH4_Error.ErrorPriority > 100 OR CH4_Error.ErrorPriority = 0     THEN CH4_Error.ErrorPriority := 100;    END_IF      END_IF
        IF wCh4_Status.4    THEN    CH4_Error.sErrorMessage := CONCAT(CH4_Error.sErrorMessage, 'Limit 2; ');                IF CH4_Error.ErrorPriority > 100 OR CH4_Error.ErrorPriority = 0     THEN CH4_Error.ErrorPriority := 100;    END_IF      END_IF
        IF wCh4_Status.6    THEN    CH4_Error.sErrorMessage := CONCAT(CH4_Error.sErrorMessage, 'Error; ');                  IF CH4_Error.ErrorPriority > 10  OR CH4_Error.ErrorPriority = 0     THEN CH4_Error.ErrorPriority := 10;     END_IF      END_IF
        IF wCh4_Status.13   THEN    CH4_Error.sErrorMessage := CONCAT(CH4_Error.sErrorMessage, 'Sync error; ');             IF CH4_Error.ErrorPriority > 10  OR CH4_Error.ErrorPriority = 0     THEN CH4_Error.ErrorPriority := 10;     END_IF      END_IF
        CH4_Error.bError := TRUE;
    ELSE
        CH4_Error.bError        := FALSE;
        CH4_Error.sErrorMessage := '';
    END_IF

    //Channel #5 Status
    IF (wCh5_Status AND 16#2057) <> 0 THEN
        CH5_Error.sErrorMessage := 'EL3255 Channel #5: ';
        IF wCH5_Status.0    THEN    CH5_Error.sErrorMessage := CONCAT(CH5_Error.sErrorMessage, 'Underrange; ');             IF CH5_Error.ErrorPriority > 100 OR CH5_Error.ErrorPriority = 0     THEN CH5_Error.ErrorPriority := 100;    END_IF      END_IF
        IF wCH5_Status.1    THEN    CH5_Error.sErrorMessage := CONCAT(CH5_Error.sErrorMessage, 'Overrange; ');              IF CH5_Error.ErrorPriority > 100 OR CH5_Error.ErrorPriority = 0     THEN CH5_Error.ErrorPriority := 100;    END_IF      END_IF
        IF wCh5_Status.2    THEN    CH5_Error.sErrorMessage := CONCAT(CH5_Error.sErrorMessage, 'Limit 1; ');                IF CH5_Error.ErrorPriority > 100 OR CH5_Error.ErrorPriority = 0     THEN CH5_Error.ErrorPriority := 100;    END_IF      END_IF
        IF wCh5_Status.4    THEN    CH5_Error.sErrorMessage := CONCAT(CH5_Error.sErrorMessage, 'Limit 2; ');                IF CH5_Error.ErrorPriority > 100 OR CH5_Error.ErrorPriority = 0     THEN CH5_Error.ErrorPriority := 100;    END_IF      END_IF
        IF wCh5_Status.6    THEN    CH5_Error.sErrorMessage := CONCAT(CH5_Error.sErrorMessage, 'Error; ');                  IF CH5_Error.ErrorPriority > 10  OR CH5_Error.ErrorPriority = 0     THEN CH5_Error.ErrorPriority := 10;     END_IF      END_IF
        IF wCh5_Status.13   THEN    CH5_Error.sErrorMessage := CONCAT(CH5_Error.sErrorMessage, 'Sync error; ');             IF CH5_Error.ErrorPriority > 10  OR CH5_Error.ErrorPriority = 0     THEN CH5_Error.ErrorPriority := 10;     END_IF      END_IF
        CH5_Error.bError := TRUE;
    ELSE
        CH5_Error.bError        := FALSE;
        CH5_Error.sErrorMessage := '';
    END_IF

END_IF

//Error FB instance
EL3255_Error(
    En                  := TRUE,
    iTerminal_ID        := iTerminal_ID,
    bWcState            := WcState_WcState,
    uiInfoData_State    := InfoData_State,
    pErrorSystem        := ErrorSystem,
    bError              => bError,
);

CH1_Error (
    En              := En,
    bError          := ,
    sErrorMessage   := ,
    ErrorPriority   := ,
    iTerminal_ID    := iTerminal_ID,
    pErrorSystem    := ErrorSystem,
    EnO             => ,
);

CH2_Error (
    En              := En,
    bError          := ,
    sErrorMessage   := ,
    ErrorPriority   := ,
    iTerminal_ID    := iTerminal_ID,
    pErrorSystem    := ErrorSystem,
    EnO             => ,
);

CH3_Error (
    En              := En,
    bError          := ,
    sErrorMessage   := ,
    ErrorPriority   := ,
    iTerminal_ID    := iTerminal_ID,
    pErrorSystem    := ErrorSystem,
    EnO             => ,
);

CH4_Error (
    En              := En,
    bError          := ,
    sErrorMessage   := ,
    ErrorPriority   := ,
    iTerminal_ID    := iTerminal_ID,
    pErrorSystem    := ErrorSystem,
    EnO             => ,
);

CH5_Error (
    En              := En,
    bError          := ,
    sErrorMessage   := ,
    ErrorPriority   := ,
    iTerminal_ID    := iTerminal_ID,
    pErrorSystem    := ErrorSystem,
    EnO             => ,
);

END_FUNCTION_BLOCK

// ---- POUs/Common/Hardware/EtherCAT_Terminals/Analog_Inputs/El3742.TcPOU
//EL3742 | 2-channel analog input terminal 0…20 mA, differential input, with oversampling
FUNCTION_BLOCK El3742

VAR_INPUT
    En: BOOL;
    iTerminal_ID : INT;
    ErrorSystem : POINTER TO ST_ErrorSystem;
END_VAR

VAR_OUTPUT
    EnO: BOOL;
    bError: BOOL;
	sErrorMessage : STRING;
END_VAR

VAR
    WcState_WcState AT %I* : BOOL := FALSE;
    InfoData_State  AT %I* : UINT := 0;

    //FB-s
    EL3742_Error    : FB_TerminalError;
END_VAR

(*
* TODO: Test on hardware
*)

EnO:=En;

EL3742_Error(
    En := TRUE,
    iTerminal_ID := iTerminal_ID,
    bWcState := FALSE,
    uiInfoData_State := InfoData_State,
    pErrorSystem := ErrorSystem,
    bError => bError,
);

IF bError THEN
	sErrorMessage:=EL3742_Error.ErrorData.sErrorMessage;
ELSE
	sErrorMessage:='';
END_IF

END_FUNCTION_BLOCK

// ---- POUs/Common/Hardware/EtherCAT_Terminals/Digital_Inputs/EL1008.TcPOU
///EL1008 | 8-channel digital input terminal 24 V DC, 3 ms
FUNCTION_BLOCK EL1008

VAR_INPUT
    En              : BOOL;
    iTerminal_ID    : INT;
    ErrorSystem     : POINTER TO ST_ErrorSystem;
END_VAR

VAR_OUTPUT
    EnO     : BOOL;
    bError  : BOOL;
END_VAR

VAR
    WcState_WcState     AT %I*  : BOOL;
    InfoData_State      AT %I*  : UINT;

    //FB-s
    EL1008_Error    : FB_TerminalError;
END_VAR

(*
* TODO: DONE!
*)
EnO:=En;

//Error FB instance
EL1008_Error(
    En                  := TRUE,
    iTerminal_ID        := iTerminal_ID,
    bWcState            := WcState_WcState,
    uiInfoData_State    := InfoData_State,
    pErrorSystem        := ErrorSystem,
    bError              => bError,
);

END_FUNCTION_BLOCK

// ---- POUs/Common/Hardware/EtherCAT_Terminals/Digital_Inputs/EL1018.TcPOU
///EL1018 | 8-channel digital input terminal 24 V DC, 10 µs
FUNCTION_BLOCK EL1018

VAR_INPUT
    En              : BOOL;
    iTerminal_ID    : INT;
    ErrorSystem     : POINTER TO ST_ErrorSystem;
END_VAR

VAR_OUTPUT
    EnO         : BOOL;
    bError      : BOOL;
END_VAR

VAR
    WcState_WcState     AT %I*  : BOOL;
    InfoData_State      AT %I*  : UINT;

    //FB-s
    EL1018_Error    : FB_TerminalError;
END_VAR

(*
* TODO: DONE!
*)
EnO:=En;

//Error FB instance
EL1018_Error(
    En                  := TRUE,
    iTerminal_ID        := iTerminal_ID,
    bWcState            := WcState_WcState,
    uiInfoData_State    := InfoData_State,
    pErrorSystem        := ErrorSystem,
    bError              => bError,
);

END_FUNCTION_BLOCK

// ---- POUs/Common/Hardware/EtherCAT_Terminals/Digital_Inputs/EL1808.TcPOU
///EL1808 | HD EtherCAT Terminals, 8-channel digital input 24 V DC, 3 ms, 2-wire connection
FUNCTION_BLOCK EL1808

VAR_INPUT
    En              : BOOL;
    iTerminal_ID    : INT;
    ErrorSystem     : POINTER TO ST_ErrorSystem;
END_VAR

VAR_OUTPUT
    EnO         : BOOL;
    bError      : BOOL;
END_VAR

VAR
    WcState_WcState     AT %I*  : BOOL;
    InfoData_State      AT %I*  : UINT;

    //FB-s
    EL1808_Error    : FB_TerminalError;
END_VAR

(*
* TODO: DONE!
*)
EnO:=En;

//Error FB instance
EL1808_Error(
    En                  := TRUE,
    iTerminal_ID        := iTerminal_ID,
    bWcState            := WcState_WcState,
    uiInfoData_State    := InfoData_State,
    pErrorSystem        := ErrorSystem,
    bError              => bError,
);

END_FUNCTION_BLOCK

// ---- POUs/Common/Hardware/EtherCAT_Terminals/Digital_Inputs/EL1819.TcPOU
///EL1819 | HD EtherCAT Terminals, 16-channel digital input 24 V DC, 10 µs
FUNCTION_BLOCK EL1819

VAR_INPUT
    En              : BOOL;
    iTerminal_ID    : INT;
    ErrorSystem     : POINTER TO ST_ErrorSystem;
END_VAR

VAR_OUTPUT
    EnO         : BOOL;
    bError      : BOOL;
END_VAR

VAR
    WcState_WcState     AT %I*  : BOOL;
    InfoData_State      AT %I*  : UINT;

    //FB-s
    EL1819_Error    : FB_TerminalError;
END_VAR

(*
* TODO: DONE!
*)
EnO:=En;

//Error FB instance
EL1819_Error(
    En                  := TRUE,
    iTerminal_ID        := iTerminal_ID,
    bWcState            := WcState_WcState,
    uiInfoData_State    := InfoData_State,
    pErrorSystem        := ErrorSystem,
    bError              => bError,
);

END_FUNCTION_BLOCK

// ---- POUs/Common/Hardware/EtherCAT_Terminals/Digital_Outputs/EL2014.TcPOU
// EL2014 | 4-channel output terminal, 24V DC, 0.5A, 4 x 0V contact
FUNCTION_BLOCK EL2014
VAR_INPUT
    En              : BOOL;
    iTerminal_ID    : INT;
    ErrorSystem     : POINTER TO ST_ErrorSystem;
END_VAR

VAR_OUTPUT
    EnO         : BOOL;
    bError      : BOOL;
END_VAR

VAR
    //Channel Diagnostic Inputs
    wCH1_Diag       AT %I*  : BYTE;
    wCH2_Diag       AT %I*  : BYTE;
    wCH3_Diag       AT %I*  : BYTE;
    wCH4_Diag       AT %I*  : BYTE;
    //Device Diagnostic Inputs
    wDevice_Diag        AT %I*  : BYTE;
    //Device State Inputs
    WcState_WcState     AT %I*  : BOOL;
    InfoData_State      AT %I*  : UINT;


    //FB-s
    EL2014_Error    : FB_TerminalError;
    CH1_Error       : FB_GenericError;
    CH2_Error       : FB_GenericError;
    CH3_Error       : FB_GenericError;
    CH4_Error       : FB_GenericError;
    DEV_Error       : FB_GenericError;
END_VAR

(*
*   TODO: Test on hardware
*)
EnO:=En;

IF En THEN

    //Channel #1 Diag
    IF wCH1_Diag <> 0 THEN
        CH1_Error.sErrorMessage := 'EL2014 Channel #1: ';
        IF wCH1_Diag.0  THEN    CH1_Error.sErrorMessage := CONCAT(CH1_Error.sErrorMessage, 'Overtemperature; ');            IF CH1_Error.ErrorPriority > 10  OR CH1_Error.ErrorPriority = 0     THEN CH1_Error.ErrorPriority := 10;     END_IF      END_IF
        IF wCH1_Diag.1  THEN    CH1_Error.sErrorMessage := CONCAT(CH1_Error.sErrorMessage, 'Open Load; ');                  IF CH1_Error.ErrorPriority > 100 OR CH1_Error.ErrorPriority = 0     THEN CH1_Error.ErrorPriority := 100;    END_IF      END_IF
        IF wCH1_Diag.2  THEN    CH1_Error.sErrorMessage := CONCAT(CH1_Error.sErrorMessage, 'Overcurrent; ');                IF CH1_Error.ErrorPriority > 10  OR CH1_Error.ErrorPriority = 0     THEN CH1_Error.ErrorPriority := 10;     END_IF      END_IF
        IF wCH1_Diag.3  THEN    CH1_Error.sErrorMessage := CONCAT(CH1_Error.sErrorMessage, 'Short Circuit to 24V; ');       IF CH1_Error.ErrorPriority > 10  OR CH1_Error.ErrorPriority = 0     THEN CH1_Error.ErrorPriority := 10;     END_IF      END_IF
        CH1_Error.bError := TRUE;
    ELSE
        CH1_Error.bError := FALSE;
        CH1_Error.sErrorMessage := '';
    END_IF

    //Channel #2 Diag
    IF wCH2_Diag <> 0 THEN
        CH2_Error.sErrorMessage := 'EL2014 Channel #2: ';
        IF wCH2_Diag.0  THEN    CH2_Error.sErrorMessage := CONCAT(CH2_Error.sErrorMessage, 'Overtemperature; ');            IF CH2_Error.ErrorPriority > 10  OR CH2_Error.ErrorPriority = 0     THEN CH2_Error.ErrorPriority := 10;     END_IF      END_IF
        IF wCH2_Diag.1  THEN    CH2_Error.sErrorMessage := CONCAT(CH2_Error.sErrorMessage, 'Open Load; ');                  IF CH2_Error.ErrorPriority > 100 OR CH2_Error.ErrorPriority = 0     THEN CH2_Error.ErrorPriority := 100;    END_IF      END_IF
        IF wCH2_Diag.2  THEN    CH2_Error.sErrorMessage := CONCAT(CH2_Error.sErrorMessage, 'Overcurrent; ');                IF CH2_Error.ErrorPriority > 10  OR CH2_Error.ErrorPriority = 0     THEN CH2_Error.ErrorPriority := 10;     END_IF      END_IF
        IF wCH2_Diag.3  THEN    CH2_Error.sErrorMessage := CONCAT(CH2_Error.sErrorMessage, 'Short Circuit to 24V; ');       IF CH2_Error.ErrorPriority > 10  OR CH2_Error.ErrorPriority = 0     THEN CH2_Error.ErrorPriority := 10;     END_IF      END_IF
        CH2_Error.bError := TRUE;
    ELSE
        CH2_Error.bError := FALSE;
        CH2_Error.sErrorMessage := '';
    END_IF

    //Channel #3 Diag
    IF wCH3_Diag <> 0 THEN
        CH3_Error.sErrorMessage := 'EL2014 Channel #3: ';
        IF wCH3_Diag.0  THEN    CH3_Error.sErrorMessage := CONCAT(CH3_Error.sErrorMessage, 'Overtemperature; ');            IF CH3_Error.ErrorPriority > 10  OR CH3_Error.ErrorPriority = 0     THEN CH3_Error.ErrorPriority := 10;     END_IF      END_IF
        IF wCH3_Diag.1  THEN    CH3_Error.sErrorMessage := CONCAT(CH3_Error.sErrorMessage, 'Open Load; ');                  IF CH3_Error.ErrorPriority > 100 OR CH3_Error.ErrorPriority = 0     THEN CH3_Error.ErrorPriority := 100;    END_IF      END_IF
        IF wCH3_Diag.2  THEN    CH3_Error.sErrorMessage := CONCAT(CH3_Error.sErrorMessage, 'Overcurrent; ');                IF CH3_Error.ErrorPriority > 10  OR CH3_Error.ErrorPriority = 0     THEN CH3_Error.ErrorPriority := 10;     END_IF      END_IF
        IF wCH3_Diag.3  THEN    CH3_Error.sErrorMessage := CONCAT(CH3_Error.sErrorMessage, 'Short Circuit to 24V; ');       IF CH3_Error.ErrorPriority > 10  OR CH3_Error.ErrorPriority = 0     THEN CH3_Error.ErrorPriority := 10;     END_IF      END_IF
        CH3_Error.bError := TRUE;
    ELSE
        CH3_Error.bError := FALSE;
        CH3_Error.sErrorMessage := '';
    END_IF

    //Channel #4 Diag
    IF wCH4_Diag <> 0 THEN
        CH4_Error.sErrorMessage := 'EL2014 Channel #4: ';
        IF wCH4_Diag.0  THEN    CH4_Error.sErrorMessage := CONCAT(CH4_Error.sErrorMessage, 'Overtemperature; ');            IF CH4_Error.ErrorPriority > 10  OR CH4_Error.ErrorPriority = 0     THEN CH4_Error.ErrorPriority := 10;     END_IF      END_IF
        IF wCH4_Diag.1  THEN    CH4_Error.sErrorMessage := CONCAT(CH4_Error.sErrorMessage, 'Open Load; ');                  IF CH4_Error.ErrorPriority > 100 OR CH4_Error.ErrorPriority = 0     THEN CH4_Error.ErrorPriority := 100;    END_IF      END_IF
        IF wCH4_Diag.2  THEN    CH4_Error.sErrorMessage := CONCAT(CH4_Error.sErrorMessage, 'Overcurrent; ');                IF CH4_Error.ErrorPriority > 10  OR CH4_Error.ErrorPriority = 0     THEN CH4_Error.ErrorPriority := 10;     END_IF      END_IF
        IF wCH4_Diag.3  THEN    CH4_Error.sErrorMessage := CONCAT(CH4_Error.sErrorMessage, 'Short Circuit to 24V; ');       IF CH4_Error.ErrorPriority > 10  OR CH4_Error.ErrorPriority = 0     THEN CH4_Error.ErrorPriority := 10;     END_IF      END_IF
        CH4_Error.bError := TRUE;
    ELSE
        CH4_Error.bError := FALSE;
        CH4_Error.sErrorMessage := '';
    END_IF

    //Device Diag
    IF wDevice_Diag <> 0 THEN
        DEV_Error.sErrorMessage := 'EL2014: ' ;
        IF wDevice_Diag.0   THEN    DEV_Error.sErrorMessage := CONCAT(DEV_Error.sErrorMessage, 'Common Fault; ');                   IF DEV_Error.ErrorPriority > 100 OR DEV_Error.ErrorPriority = 0     THEN DEV_Error.ErrorPriority := 100;    END_IF      END_IF
        IF wDevice_Diag.1   THEN    DEV_Error.sErrorMessage := CONCAT(DEV_Error.sErrorMessage, 'Device Overtemperature; ');         IF DEV_Error.ErrorPriority > 10  OR DEV_Error.ErrorPriority = 0     THEN DEV_Error.ErrorPriority := 10;     END_IF      END_IF
        IF wDevice_Diag.2   THEN    DEV_Error.sErrorMessage := CONCAT(DEV_Error.sErrorMessage, 'Undervoltage; ');                   IF DEV_Error.ErrorPriority > 10  OR DEV_Error.ErrorPriority = 0     THEN DEV_Error.ErrorPriority := 10;     END_IF      END_IF
        IF wDevice_Diag.3   THEN    DEV_Error.sErrorMessage := CONCAT(DEV_Error.sErrorMessage, 'Missing Voltage; ');                IF DEV_Error.ErrorPriority > 10  OR DEV_Error.ErrorPriority = 0     THEN DEV_Error.ErrorPriority := 10;     END_IF      END_IF
        DEV_Error.bError := TRUE;
    ELSE
        DEV_Error.bError := FALSE;
        DEV_Error.sErrorMessage := '';
    END_IF

END_IF

//Terminal's State of Operation
EL2014_Error(
    En                  := TRUE,
    iTerminal_ID        := iTerminal_ID,
    bWcState            := WcState_WcState,
    uiInfoData_State    := InfoData_State,
    pErrorSystem        := ErrorSystem,
    bError              => bError,
);

CH1_Error (
    En                  :=  En,
    bError              :=  ,
    sErrorMessage       :=  ,
    ErrorPriority       :=  ,
    iTerminal_ID        :=  iTerminal_ID,
    pErrorSystem        :=  ErrorSystem,
    EnO                 =>  ,
);

CH2_Error (
    En                  :=  En,
    bError              :=  ,
    sErrorMessage       :=  ,
    ErrorPriority       :=  ,
    iTerminal_ID        :=  iTerminal_ID,
    pErrorSystem        :=  ErrorSystem,
    EnO                 =>  ,
);

CH3_Error (
    En                  :=  En,
    bError              :=  ,
    sErrorMessage       :=  ,
    ErrorPriority       :=  ,
    iTerminal_ID        :=  iTerminal_ID,
    pErrorSystem        :=  ErrorSystem,
    EnO                 =>  ,
);

CH4_Error (
    En                  :=  En,
    bError              :=  ,
    sErrorMessage       :=  ,
    ErrorPriority       :=  ,
    iTerminal_ID        :=  iTerminal_ID,
    pErrorSystem        :=  ErrorSystem,
    EnO                 =>  ,
);

DEV_Error (
    En                  :=  En,
    bError              :=  ,
    sErrorMessage       :=  ,
    ErrorPriority       :=  ,
    iTerminal_ID        :=  iTerminal_ID,
    pErrorSystem        :=  ErrorSystem,
    EnO                 =>  ,
);

END_FUNCTION_BLOCK

// ---- POUs/Common/Hardware/EtherCAT_Terminals/Digital_Outputs/EL2252.TcPOU
///EL2252 | XFC, 2-channel digital output terminal with time stamp, tri-state
FUNCTION_BLOCK EL2252
VAR_INPUT
    En              : BOOL;
    iTerminal_ID    : INT;
    ErrorSystem     : POINTER TO ST_ErrorSystem;
END_VAR

VAR_OUTPUT
    EnO     : BOOL;
    bError  : BOOL;
END_VAR

VAR
    WcState_WcState     AT %I*: BOOL;
    InfoData_State      AT %I*: UINT;

    //FB-s
    EL2252_Error    : FB_TerminalError;
END_VAR

(*
* TODO: DONE!
*)

EL2252_Error(
    En                  := TRUE,
    iTerminal_ID        := iTerminal_ID,
    bWcState            := WcState_WcState,
    uiInfoData_State    := InfoData_State,
    pErrorSystem        := ErrorSystem,
    bError              => bError,
);

END_FUNCTION_BLOCK

// ---- POUs/Common/Hardware/EtherCAT_Terminals/Digital_Outputs/EL2808.TcPOU
FUNCTION_BLOCK EL2808

VAR_INPUT
    En              : BOOL;
    iTerminal_ID    : INT;
    ErrorSystem     : POINTER TO ST_ErrorSystem;
END_VAR

VAR_OUTPUT
    EnO     : BOOL;
    bError  : BOOL;
END_VAR

VAR
    WcState_WcState     AT %I*  : BOOL;
    InfoData_State      AT %I*  : UINT;

    //FB-s
    EL2808_Error    : FB_TerminalError;
END_VAR

(*
* TODO: DONE!
*)
EnO:=En;

EL2808_Error(
    En                  := TRUE,
    iTerminal_ID        := iTerminal_ID,
    bWcState            := WcState_WcState,
    uiInfoData_State    := InfoData_State,
    pErrorSystem        := ErrorSystem,
    bError              => bError,
);

END_FUNCTION_BLOCK

// ---- POUs/Common/Hardware/EtherCAT_Terminals/Drives/EL2522.TcPOU
//EL2522 | 2-channel Puls/Dir terminal
FUNCTION_BLOCK EL2522

VAR_INPUT
    En: BOOL;
    iTerminal_ID : INT;
    ErrorSystem : POINTER TO ST_ErrorSystem;
END_VAR

VAR_OUTPUT
    EnO: BOOL;
    bError: BOOL;
END_VAR

VAR
    //WC_State is handled by NC, so NOT included here.
    InfoData_State AT %I*: UINT;

    //FB-s
    EL2522_Error    : FB_TerminalError;
END_VAR

(*
* TODO: Test on hardware
*)

EnO:=En;

EL2522_Error(
    En := TRUE,
    iTerminal_ID := iTerminal_ID,
    bWcState := FALSE,
    uiInfoData_State := InfoData_State,
    pErrorSystem := ErrorSystem,
    bError => bError,
);

END_FUNCTION_BLOCK

// ---- POUs/Common/Hardware/EtherCAT_Terminals/Drives/EL4134.TcPOU
//EL4134 | 4-channel analog output terminal, -10..+10V, 16 bit
FUNCTION_BLOCK EL4134

VAR_INPUT
    En: BOOL;
    iTerminal_ID : INT;
    ErrorSystem : POINTER TO ST_ErrorSystem;
END_VAR

VAR_OUTPUT
    EnO: BOOL;
    bError: BOOL;
END_VAR

VAR
    //WC_State is handled by NC, so NOT included here.
    InfoData_State AT %I*: UINT;

    //FB-s
    EL4134_Error    : FB_TerminalError;
END_VAR

(*
* TODO: Test on hardware
*)

EnO:=En;

EL4134_Error(
    En := TRUE,
    iTerminal_ID := iTerminal_ID,
    bWcState := FALSE,
    uiInfoData_State := InfoData_State,
    pErrorSystem := ErrorSystem,
    bError => bError,
);

END_FUNCTION_BLOCK

// ---- POUs/Common/Hardware/EtherCAT_Terminals/Drives/EL7037.TcPOU
//EL7037 | Stepper motor terminal, 24V DC, 1.5A
FUNCTION_BLOCK EL7037

VAR_INPUT
    En: BOOL;
    iTerminal_ID : INT;
    ErrorSystem : POINTER TO ST_ErrorSystem;
END_VAR

VAR_OUTPUT
    EnO: BOOL;
    bError: BOOL;
END_VAR

VAR
    //WC_State is handled by NC, so NOT included here.
    InfoData_State AT %I*: UINT;

    //FB-s
    EL7037_Error    : FB_TerminalError;
END_VAR

(*
* TODO: Test on hardware
*)

EnO:=En;

EL7037_Error(
    En := TRUE,
    iTerminal_ID := iTerminal_ID,
    bWcState := FALSE,
    uiInfoData_State := InfoData_State,
    pErrorSystem := ErrorSystem,
    bError => bError,
);

END_FUNCTION_BLOCK

// ---- POUs/Common/Hardware/EtherCAT_Terminals/Drives/EL7041_0052.TcPOU
//EL7041-0052 | Stepper motor terminal, 50V DC, 5A
FUNCTION_BLOCK EL7041_0052

VAR_INPUT
    En: BOOL;
    iTerminal_ID : INT;
    ErrorSystem : POINTER TO ST_ErrorSystem;
END_VAR

VAR_OUTPUT
    EnO: BOOL;
    bError: BOOL;
END_VAR

VAR
    //WC_State is handled by NC, so NOT included here.
    InfoData_State AT %I*: UINT;

    //FB-s
    EL7041_Error    : FB_TerminalError;
END_VAR

(*
* TODO: Test on hardware
*)

EnO:=En;

EL7041_Error(
    En := TRUE,
    iTerminal_ID := iTerminal_ID,
    bWcState := FALSE,
    uiInfoData_State := InfoData_State,
    pErrorSystem := ErrorSystem,
    bError => bError,
);

END_FUNCTION_BLOCK

// ---- POUs/Common/Hardware/EtherCAT_Terminals/Drives/EL7047.TcPOU
//EL7037 | Stepper motor terminal, 50V DC, 5A, Vector Control, Incremental Encoder
FUNCTION_BLOCK EL7047

VAR_INPUT
    En: BOOL;
    iTerminal_ID : INT;
    ErrorSystem : POINTER TO ST_ErrorSystem;
END_VAR

VAR_OUTPUT
    EnO: BOOL;
    bError: BOOL;
END_VAR

VAR
    //WC_State is handled by NC, so NOT included here.
    InfoData_State AT %I*: UINT;

    //FB-s
    EL7047_Error    : FB_TerminalError;
END_VAR

EnO:=En;

EL7047_Error(
    En := TRUE,
    iTerminal_ID := iTerminal_ID,
    bWcState := FALSE,
    uiInfoData_State := InfoData_State,
    pErrorSystem := ErrorSystem,
    bError => bError,
);

END_FUNCTION_BLOCK

// ---- POUs/Common/Hardware/EtherCAT_Terminals/Drives/EL7211.TcPOU
//EL7211 | Servo terminal, for resolver, 50V DC, 4.5Arms
FUNCTION_BLOCK EL7211

VAR_INPUT
    En: BOOL;
    iTerminal_ID : INT;
    ErrorSystem : POINTER TO ST_ErrorSystem;
END_VAR

VAR_OUTPUT
    EnO: BOOL;
    bError: BOOL;
END_VAR

VAR
    WcState_WcState AT %I* : BOOL := FALSE;
    InfoData_State  AT %I* : UINT := 0;

    //FB-s
    EL7211_Error    : FB_TerminalError;
END_VAR

(*
* TODO: Test on hardware
*)

EnO:=En;

EL7211_Error(
    En := TRUE,
    iTerminal_ID := iTerminal_ID,
    bWcState := FALSE,
    uiInfoData_State := InfoData_State,
    pErrorSystem := ErrorSystem,
    bError => bError,
);

END_FUNCTION_BLOCK

// ---- POUs/Common/Hardware/EtherCAT_Terminals/Feedback_Terminals/EL5002.TcPOU
//EL5002 | 2-chennel SSI absolute encoder terminal
FUNCTION_BLOCK EL5002

VAR_INPUT
    En: BOOL;
    iTerminal_ID : INT;
    ErrorSystem : POINTER TO ST_ErrorSystem;
END_VAR

VAR_OUTPUT
    EnO: BOOL;
    bError: BOOL;
END_VAR

VAR
    //WC_State is handled by NC, so NOT included here.
    InfoData_State AT %I*: UINT;

    //FB-s
    EL5002_Error    : FB_TerminalError;
END_VAR

(*
* TODO: Test on hardware
*)

EnO:=En;

EL5002_Error(
    En := TRUE,
    iTerminal_ID := iTerminal_ID,
    bWcState := FALSE,
    uiInfoData_State := InfoData_State,
    pErrorSystem := ErrorSystem,
    bError => bError,
);

END_FUNCTION_BLOCK

// ---- POUs/Common/Hardware/EtherCAT_Terminals/Feedback_Terminals/EL5042.TcPOU
//EL5042 | 2-channel BiSS-C absolute encoder terminal
FUNCTION_BLOCK EL5042

VAR_INPUT
    En: BOOL;
    iTerminal_ID    : INT;
    ErrorSystem     : POINTER TO ST_ErrorSystem;
END_VAR

VAR_OUTPUT
    EnO     : BOOL;
    bError  : BOOL;
END_VAR

VAR
    //WC_State is handled by NC, so NOT included here.
    InfoData_State      AT %I*  : UINT;

    //FB-s
    EL5042_Error    : FB_TerminalError;
END_VAR

(*
* TODO: Test on hardware
*)
EnO:=En;

//Error FB instances
EL5042_Error(
    En := TRUE,
    iTerminal_ID := iTerminal_ID,
    bWcState := FALSE,
    uiInfoData_State := InfoData_State,
    pErrorSystem := ErrorSystem,
    bError => bError,
);

END_FUNCTION_BLOCK

// ---- POUs/Common/Hardware/EtherCAT_Terminals/Feedback_Terminals/EL5101.TcPOU
// EL5101 | 1-channel incremental encoder terminal, 5V, RS422
FUNCTION_BLOCK EL5101

VAR_INPUT
    En              : BOOL;
    iTerminal_ID    : INT;
    ErrorSystem     : POINTER TO ST_ErrorSystem;
END_VAR

VAR_OUTPUT
    EnO     : BOOL;
    bError  : BOOL;
END_VAR

VAR
    //WC_State is handled by NC, so NOT included here.
    InfoData_State      AT %I* : UINT;

    //FB-s
    EL5101_Error    : FB_TerminalError;
END_VAR

(*
* TODO: Channel Status word (Connected to NC -> Not needed )
*)
EnO:=En;

//Error FB instances
EL5101_Error(
    En                  := TRUE,
    iTerminal_ID        := iTerminal_ID,
    bWcState            := FALSE,
    uiInfoData_State    := InfoData_State,
    pErrorSystem        := ErrorSystem,
    bError              => bError,
);

END_FUNCTION_BLOCK

// ---- POUs/Common/Hardware/EtherCAT_Terminals/System/EK1100.TcPOU
FUNCTION_BLOCK EK1100

VAR_INPUT
    En              : BOOL;
    iTerminal_ID    : INT;
    ErrorSystem     : POINTER TO ST_ErrorSystem;
END_VAR

VAR_OUTPUT
    EnO     : BOOL;
    bError  : BOOL;
	sErrorMessage       : STRING;
END_VAR

VAR
    InfoData_State  AT %I*  : UINT;

    //FB-s
    EK1100_Error    : FB_TerminalError;
END_VAR

(*
* TODO: DONE!
*)
EnO:=En;

